   1:  PR[GP1:91,1] = PR[GP1:90,1] + 57.997;
   1:  PR[GP1:91,2] = PR[GP1:90,2] + 23.981;
   1:L PR[91] R[100]mm/sec CNT100;
   1:  PR[GP1:91,1] = PR[GP1:90,1] + 53.597;
   1:  PR[GP1:91,2] = PR[GP1:90,2] + 27.915;
   1:L PR[91] R[100]mm/sec CNT100;
   1:  PR[GP1:91,1] = PR[GP1:90,1] + 52.373;
   1:  PR[GP1:91,2] = PR[GP1:90,2] + 28.903;
   1:L PR[91] R[100]mm/sec CNT100;
   1:  PR[GP1:91,1] = PR[GP1:90,1] + 47.316;
   1:  PR[GP1:91,2] = PR[GP1:90,2] + 32.038;
   1:L PR[91] R[100]mm/sec CNT100;
   1:  PR[GP1:91,1] = PR[GP1:90,1] + 42.338;
   1:  PR[GP1:91,2] = PR[GP1:90,2] + 34.026;
   1:L PR[91] R[100]mm/sec CNT100;
   1:  PR[GP1:91,1] = PR[GP1:90,1] + 39.377;
   1:  PR[GP1:91,2] = PR[GP1:90,2] + 35.072;
   1:L PR[91] R[100]mm/sec CNT100;
   1:  PR[GP1:91,1] = PR[GP1:90,1] + 34.292;
   1:  PR[GP1:91,2] = PR[GP1:90,2] + 36.166;
   1:L PR[91] R[100]mm/sec CNT100;
   1:  PR[GP1:91,1] = PR[GP1:90,1] + 29.702;
   1:  PR[GP1:91,2] = PR[GP1:90,2] + 36.339;
   1:L PR[91] R[100]mm/sec CNT100;
   1:  PR[GP1:91,1] = PR[GP1:90,1] + 24.959;
   1:  PR[GP1:91,2] = PR[GP1:90,2] + 36.356;
   1:L PR[91] R[100]mm/sec CNT100;
   1:  PR[GP1:91,1] = PR[GP1:90,1] + 20.626;
   1:  PR[GP1:91,2] = PR[GP1:90,2] + 35.786;
   1:L PR[91] R[100]mm/sec CNT100;
   1:  PR[GP1:91,1] = PR[GP1:90,1] + 16.906;
   1:  PR[GP1:91,2] = PR[GP1:90,2] + 34.602;
   1:L PR[91] R[100]mm/sec CNT100;
   1:  PR[GP1:91,1] = PR[GP1:90,1] + 11.165;
   1:  PR[GP1:91,2] = PR[GP1:90,2] + 32.612;
   1:L PR[91] R[100]mm/sec CNT100;
   1:  PR[GP1:91,1] = PR[GP1:90,1] + 7.980;
   1:  PR[GP1:91,2] = PR[GP1:90,2] + 30.950;
   1:L PR[91] R[100]mm/sec CNT100;
   1:  PR[GP1:91,1] = PR[GP1:90,1] + 5.211;
   1:  PR[GP1:91,2] = PR[GP1:90,2] + 28.994;
   1:L PR[91] R[100]mm/sec CNT100;
   1:  PR[GP1:91,1] = PR[GP1:90,1] + 4.255;
   1:  PR[GP1:91,2] = PR[GP1:90,2] + 28.246;
   1:L PR[91] R[100]mm/sec CNT100;
   1:  PR[GP1:91,1] = PR[GP1:90,1] + 3.446;
   1:  PR[GP1:91,2] = PR[GP1:90,2] + 27.305;
   1:L PR[91] R[100]mm/sec CNT100;
   1:  PR[GP1:91,1] = PR[GP1:90,1] + 1.713;
   1:  PR[GP1:91,2] = PR[GP1:90,2] + 26.621;
   1:L PR[91] R[100]mm/sec CNT100;
   1:  PR[GP1:91,1] = PR[GP1:90,1] + 1.290;
   1:  PR[GP1:91,2] = PR[GP1:90,2] + 26.404;
   1:L PR[91] R[100]mm/sec CNT100;
   1:  ! -- Layer/Ebene 89 -- !;
   1:  PR[91] = PR[90];
   1:  PR[GP1:91,1] = PR[GP1:90,1] + -2.453;
   1:  PR[GP1:91,2] = PR[GP1:90,2] + 27.220;
   1:  PR[GP1:91,3] = PR[GP1:90,3] + 54.595;
   1:L PR[91] R[100]mm/sec CNT100;
   1:  PR[GP1:91,1] = PR[GP1:90,1] + -3.226;
   1:  PR[GP1:91,2] = PR[GP1:90,2] + 27.613;
   1:L PR[91] R[100]mm/sec CNT100;
   1:  PR[GP1:91,1] = PR[GP1:90,1] + -3.881;
   1:  PR[GP1:91,2] = PR[GP1:90,2] + 28.375;
   1:L PR[91] R[100]mm/sec CNT100;
   1:  PR[GP1:91,1] = PR[GP1:90,1] + -4.669;
   1:  PR[GP1:91,2] = PR[GP1:90,2] + 28.992;
   1:L PR[91] R[100]mm/sec CNT100;
   1:  PR[GP1:91,1] = PR[GP1:90,1] + -7.549;
   1:  PR[GP1:91,2] = PR[GP1:90,2] + 31.027;
   1:L PR[91] R[100]mm/sec CNT100;
   1:  PR[GP1:91,1] = PR[GP1:90,1] + -10.616;
   1:  PR[GP1:91,2] = PR[GP1:90,2] + 32.632;
   1:L PR[91] R[100]mm/sec CNT100;
   1:  PR[GP1:91,1] = PR[GP1:90,1] + -14.394;
   1:  PR[GP1:91,2] = PR[GP1:90,2] + 33.846;
   1:L PR[91] R[100]mm/sec CNT100;
   1:  PR[GP1:91,1] = PR[GP1:90,1] + -20.227;
   1:  PR[GP1:91,2] = PR[GP1:90,2] + 35.862;
   1:L PR[91] R[100]mm/sec CNT100;
   1:  PR[GP1:91,1] = PR[GP1:90,1] + -24.397;
   1:  PR[GP1:91,2] = PR[GP1:90,2] + 36.407;
   1:L PR[91] R[100]mm/sec CNT100;
   1:  PR[GP1:91,1] = PR[GP1:90,1] + -29.289;
   1:  PR[GP1:91,2] = PR[GP1:90,2] + 36.239;
   1:L PR[91] R[100]mm/sec CNT100;
   1:  PR[GP1:91,1] = PR[GP1:90,1] + -33.933;
   1:  PR[GP1:91,2] = PR[GP1:90,2] + 36.216;
   1:L PR[91] R[100]mm/sec CNT100;
   1:  PR[GP1:91,1] = PR[GP1:90,1] + -38.847;
   1:  PR[GP1:91,2] = PR[GP1:90,2] + 35.155;
   1:L PR[91] R[100]mm/sec CNT100;
   1:  PR[GP1:91,1] = PR[GP1:90,1] + -44.230;
   1:  PR[GP1:91,2] = PR[GP1:90,2] + 33.024;
   1:L PR[91] R[100]mm/sec CNT100;
   1:  PR[GP1:91,1] = PR[GP1:90,1] + -46.959;
   1:  PR[GP1:91,2] = PR[GP1:90,2] + 32.055;
   1:L PR[91] R[100]mm/sec CNT100;
   1:  PR[GP1:91,1] = PR[GP1:90,1] + -51.884;
   1:  PR[GP1:91,2] = PR[GP1:90,2] + 28.987;
   1:L PR[91] R[100]mm/sec CNT100;
   1:  PR[GP1:91,1] = PR[GP1:90,1] + -56.664;
   1:  PR[GP1:91,2] = PR[GP1:90,2] + 24.742;
   1:L PR[91] R[100]mm/sec CNT100;
   1:  PR[GP1:91,1] = PR[GP1:90,1] + -57.689;
   1:  PR[GP1:91,2] = PR[GP1:90,2] + 23.913;
   1:L PR[91] R[100]mm/sec CNT100;
   1:  PR[GP1:91,1] = PR[GP1:90,1] + -61.507;
   1:  PR[GP1:91,2] = PR[GP1:90,2] + 18.944;
   1:L PR[91] R[100]mm/sec CNT100;
   1:  PR[GP1:91,1] = PR[GP1:90,1] + -64.708;
   1:  PR[GP1:91,2] = PR[GP1:90,2] + 12.732;
   1:L PR[91] R[100]mm/sec CNT100;
   1:  PR[GP1:91,1] = PR[GP1:90,1] + -64.834;
   1:  PR[GP1:91,2] = PR[GP1:90,2] + 12.522;
   1:L PR[91] R[100]mm/sec CNT100;
   1:  PR[GP1:91,1] = PR[GP1:90,1] + -66.655;
   1:  PR[GP1:91,2] = PR[GP1:90,2] + 6.345;
   1:L PR[91] R[100]mm/sec CNT100;
   1:  PR[GP1:91,1] = PR[GP1:90,1] + -67.234;
   1:  PR[GP1:91,2] = PR[GP1:90,2] + -0.052;
   1:L PR[91] R[100]mm/sec CNT100;
   1:  PR[GP1:91,1] = PR[GP1:90,1] + -67.229;
   1:  PR[GP1:91,2] = PR[GP1:90,2] + -0.083;
   1:L PR[91] R[100]mm/sec CNT100;
   1:  PR[GP1:91,1] = PR[GP1:90,1] + -66.655;
   1:  PR[GP1:91,2] = PR[GP1:90,2] + -6.489;
   1:L PR[91] R[100]mm/sec CNT100;
   1:  PR[GP1:91,1] = PR[GP1:90,1] + -64.828;
   1:  PR[GP1:91,2] = PR[GP1:90,2] + -12.686;
   1:L PR[91] R[100]mm/sec CNT100;
   1:  PR[GP1:91,1] = PR[GP1:90,1] + -61.862;
   1:  PR[GP1:91,2] = PR[GP1:90,2] + -18.501;
   1:L PR[91] R[100]mm/sec CNT100;
   1:  PR[GP1:91,1] = PR[GP1:90,1] + -61.519;
   1:  PR[GP1:91,2] = PR[GP1:90,2] + -19.072;
   1:L PR[91] R[100]mm/sec CNT100;
   1:  PR[GP1:91,1] = PR[GP1:90,1] + -57.679;
   1:  PR[GP1:91,2] = PR[GP1:90,2] + -24.070;
   1:L PR[91] R[100]mm/sec CNT100;
   1:  PR[GP1:91,1] = PR[GP1:90,1] + -53.369;
   1:  PR[GP1:91,2] = PR[GP1:90,2] + -27.936;
   1:L PR[91] R[100]mm/sec CNT100;
   1:  PR[GP1:91,1] = PR[GP1:90,1] + -51.894;
   1:  PR[GP1:91,2] = PR[GP1:90,2] + -29.125;
   1:L PR[91] R[100]mm/sec CNT100;
   1:  PR[GP1:91,1] = PR[GP1:90,1] + -46.946;
   1:  PR[GP1:91,2] = PR[GP1:90,2] + -32.207;
   1:L PR[91] R[100]mm/sec CNT100;
   1:  PR[GP1:91,1] = PR[GP1:90,1] + -42.112;
   1:  PR[GP1:91,2] = PR[GP1:90,2] + -34.148;
   1:L PR[91] R[100]mm/sec CNT100;
   1:  PR[GP1:91,1] = PR[GP1:90,1] + -38.854;
   1:  PR[GP1:91,2] = PR[GP1:90,2] + -35.298;
   1:L PR[91] R[100]mm/sec CNT100;
   1:  PR[GP1:91,1] = PR[GP1:90,1] + -33.917;
   1:  PR[GP1:91,2] = PR[GP1:90,2] + -36.363;
   1:L PR[91] R[100]mm/sec CNT100;
   1:  PR[GP1:91,1] = PR[GP1:90,1] + -29.447;
   1:  PR[GP1:91,2] = PR[GP1:90,2] + -36.535;
   1:L PR[91] R[100]mm/sec CNT100;
   1:  PR[GP1:91,1] = PR[GP1:90,1] + -24.397;
   1:  PR[GP1:91,2] = PR[GP1:90,2] + -36.551;
   1:L PR[91] R[100]mm/sec CNT100;
   1:  PR[GP1:91,1] = PR[GP1:90,1] + -20.210;
   1:  PR[GP1:91,2] = PR[GP1:90,2] + -36.004;
   1:L PR[91] R[100]mm/sec CNT100;
   1:  PR[GP1:91,1] = PR[GP1:90,1] + -16.625;
   1:  PR[GP1:91,2] = PR[GP1:90,2] + -34.863;
   1:L PR[91] R[100]mm/sec CNT100;
   1:  PR[GP1:91,1] = PR[GP1:90,1] + -10.613;
   1:  PR[GP1:91,2] = PR[GP1:90,2] + -32.774;
   1:L PR[91] R[100]mm/sec CNT100;
   1:  PR[GP1:91,1] = PR[GP1:90,1] + -7.546;
   1:  PR[GP1:91,2] = PR[GP1:90,2] + -31.169;
   1:L PR[91] R[100]mm/sec CNT100;
   1:  PR[GP1:91,1] = PR[GP1:90,1] + -3.573;
   1:  PR[GP1:91,2] = PR[GP1:90,2] + -28.282;
   1:L PR[91] R[100]mm/sec CNT100;
   1:  PR[GP1:91,1] = PR[GP1:90,1] + -3.414;
   1:  PR[GP1:91,2] = PR[GP1:90,2] + -28.158;
   1:L PR[91] R[100]mm/sec CNT100;
   1:  PR[GP1:91,1] = PR[GP1:90,1] + -3.168;
   1:  PR[GP1:91,2] = PR[GP1:90,2] + -27.873;
   1:L PR[91] R[100]mm/sec CNT100;
   1:  PR[GP1:91,1] = PR[GP1:90,1] + 0.870;
   1:  PR[GP1:91,2] = PR[GP1:90,2] + -27.006;
   1:L PR[91] R[100]mm/sec CNT100;
   1:  PR[GP1:91,1] = PR[GP1:90,1] + 1.216;
   1:  PR[GP1:91,2] = PR[GP1:90,2] + -26.822;
   1:L PR[91] R[100]mm/sec CNT100;
   1:  PR[GP1:91,1] = PR[GP1:90,1] + 3.432;
   1:  PR[GP1:91,2] = PR[GP1:90,2] + -27.937;
   1:L PR[91] R[100]mm/sec CNT100;
   1:  PR[GP1:91,1] = PR[GP1:90,1] + 3.626;
   1:  PR[GP1:91,2] = PR[GP1:90,2] + -28.162;
   1:L PR[91] R[100]mm/sec CNT100;
   1:  PR[GP1:91,1] = PR[GP1:90,1] + 3.783;
   1:  PR[GP1:91,2] = PR[GP1:90,2] + -28.285;
   1:L PR[91] R[100]mm/sec CNT100;
   1:  PR[GP1:91,1] = PR[GP1:90,1] + 7.766;
   1:  PR[GP1:91,2] = PR[GP1:90,2] + -31.179;
   1:L PR[91] R[100]mm/sec CNT100;
   1:  PR[GP1:91,1] = PR[GP1:90,1] + 10.807;
   1:  PR[GP1:91,2] = PR[GP1:90,2] + -32.766;
   1:L PR[91] R[100]mm/sec CNT100;
   1:  PR[GP1:91,1] = PR[GP1:90,1] + 14.586;
   1:  PR[GP1:91,2] = PR[GP1:90,2] + -33.980;
   1:L PR[91] R[100]mm/sec CNT100;
   1:  PR[GP1:91,1] = PR[GP1:90,1] + 20.426;
   1:  PR[GP1:91,2] = PR[GP1:90,2] + -36.002;
   1:L PR[91] R[100]mm/sec CNT100;
   1:  PR[GP1:91,1] = PR[GP1:90,1] + 24.591;
   1:  PR[GP1:91,2] = PR[GP1:90,2] + -36.549;
   1:L PR[91] R[100]mm/sec CNT100;
   1:  PR[GP1:91,1] = PR[GP1:90,1] + 29.460;
   1:  PR[GP1:91,2] = PR[GP1:90,2] + -36.386;
   1:L PR[91] R[100]mm/sec CNT100;
   1:  PR[GP1:91,1] = PR[GP1:90,1] + 34.110;
   1:  PR[GP1:91,2] = PR[GP1:90,2] + -36.365;
   1:L PR[91] R[100]mm/sec CNT100;
   1:  PR[GP1:91,1] = PR[GP1:90,1] + 39.017;
   1:  PR[GP1:91,2] = PR[GP1:90,2] + -35.309;
   1:L PR[91] R[100]mm/sec CNT100;
   1:  PR[GP1:91,1] = PR[GP1:90,1] + 44.407;
   1:  PR[GP1:91,2] = PR[GP1:90,2] + -33.186;
   1:L PR[91] R[100]mm/sec CNT100;
   1:  PR[GP1:91,1] = PR[GP1:90,1] + 47.142;
   1:  PR[GP1:91,2] = PR[GP1:90,2] + -32.216;
   1:L PR[91] R[100]mm/sec CNT100;
   1:  PR[GP1:91,1] = PR[GP1:90,1] + 52.036;
   1:  PR[GP1:91,2] = PR[GP1:90,2] + -29.183;
   1:L PR[91] R[100]mm/sec CNT100;
   1:  PR[GP1:91,1] = PR[GP1:90,1] + 56.791;
   1:  PR[GP1:91,2] = PR[GP1:90,2] + -24.972;
   1:L PR[91] R[100]mm/sec CNT100;
   1:  PR[GP1:91,1] = PR[GP1:90,1] + 57.825;
   1:  PR[GP1:91,2] = PR[GP1:90,2] + -24.135;
   1:L PR[91] R[100]mm/sec CNT100;
   1:  PR[GP1:91,1] = PR[GP1:90,1] + 61.682;
   1:  PR[GP1:91,2] = PR[GP1:90,2] + -19.128;
   1:L PR[91] R[100]mm/sec CNT100;
   1:  PR[GP1:91,1] = PR[GP1:90,1] + 64.892;
   1:  PR[GP1:91,2] = PR[GP1:90,2] + -12.967;
   1:L PR[91] R[100]mm/sec CNT100;
   1:  PR[GP1:91,1] = PR[GP1:90,1] + 65.020;
   1:  PR[GP1:91,2] = PR[GP1:90,2] + -12.754;
   1:L PR[91] R[100]mm/sec CNT100;
   1:  PR[GP1:91,1] = PR[GP1:90,1] + 66.839;
   1:  PR[GP1:91,2] = PR[GP1:90,2] + -6.669;
   1:L PR[91] R[100]mm/sec CNT100;
   1:  PR[GP1:91,1] = PR[GP1:90,1] + 67.449;
   1:  PR[GP1:91,2] = PR[GP1:90,2] + -0.072;
   1:L PR[91] R[100]mm/sec CNT100;
   1:  PR[GP1:91,1] = PR[GP1:90,1] + 66.839;
   1:  PR[GP1:91,2] = PR[GP1:90,2] + 6.525;
   1:L PR[91] R[100]mm/sec CNT100;
   1:  PR[GP1:91,1] = PR[GP1:90,1] + 65.015;
   1:  PR[GP1:91,2] = PR[GP1:90,2] + 12.629;
   1:L PR[91] R[100]mm/sec CNT100;
   1:  PR[GP1:91,1] = PR[GP1:90,1] + 62.040;
   1:  PR[GP1:91,2] = PR[GP1:90,2] + 18.394;
   1:L PR[91] R[100]mm/sec CNT100;
   1:  PR[GP1:91,1] = PR[GP1:90,1] + 61.694;
   1:  PR[GP1:91,2] = PR[GP1:90,2] + 18.969;
   1:L PR[91] R[100]mm/sec CNT100;
   1:  PR[GP1:91,1] = PR[GP1:90,1] + 57.816;
   1:  PR[GP1:91,2] = PR[GP1:90,2] + 24.003;
   1:L PR[91] R[100]mm/sec CNT100;
   1:  PR[GP1:91,1] = PR[GP1:90,1] + 53.529;
   1:  PR[GP1:91,2] = PR[GP1:90,2] + 27.836;
   1:L PR[91] R[100]mm/sec CNT100;
   1:  PR[GP1:91,1] = PR[GP1:90,1] + 52.050;
   1:  PR[GP1:91,2] = PR[GP1:90,2] + 29.030;
   1:L PR[91] R[100]mm/sec CNT100;
   1:  PR[GP1:91,1] = PR[GP1:90,1] + 47.134;
   1:  PR[GP1:91,2] = PR[GP1:90,2] + 32.078;
   1:L PR[91] R[100]mm/sec CNT100;
   1:  PR[GP1:91,1] = PR[GP1:90,1] + 42.293;
   1:  PR[GP1:91,2] = PR[GP1:90,2] + 34.011;
   1:L PR[91] R[100]mm/sec CNT100;
   1:  PR[GP1:91,1] = PR[GP1:90,1] + 39.032;
   1:  PR[GP1:91,2] = PR[GP1:90,2] + 35.162;
   1:L PR[91] R[100]mm/sec CNT100;
   1:  PR[GP1:91,1] = PR[GP1:90,1] + 34.105;
   1:  PR[GP1:91,2] = PR[GP1:90,2] + 36.222;
   1:L PR[91] R[100]mm/sec CNT100;
   1:  PR[GP1:91,1] = PR[GP1:90,1] + 29.656;
   1:  PR[GP1:91,2] = PR[GP1:90,2] + 36.390;
   1:L PR[91] R[100]mm/sec CNT100;
   1:  PR[GP1:91,1] = PR[GP1:90,1] + 24.608;
   1:  PR[GP1:91,2] = PR[GP1:90,2] + 36.408;
   1:L PR[91] R[100]mm/sec CNT100;
   1:  PR[GP1:91,1] = PR[GP1:90,1] + 20.428;
   1:  PR[GP1:91,2] = PR[GP1:90,2] + 35.858;
   1:L PR[91] R[100]mm/sec CNT100;
   1:  PR[GP1:91,1] = PR[GP1:90,1] + 16.838;
   1:  PR[GP1:91,2] = PR[GP1:90,2] + 34.716;
   1:L PR[91] R[100]mm/sec CNT100;
   1:  PR[GP1:91,1] = PR[GP1:90,1] + 10.823;
   1:  PR[GP1:91,2] = PR[GP1:90,2] + 32.631;
   1:L PR[91] R[100]mm/sec CNT100;
   1:  PR[GP1:91,1] = PR[GP1:90,1] + 7.768;
   1:  PR[GP1:91,2] = PR[GP1:90,2] + 31.037;
   1:L PR[91] R[100]mm/sec CNT100;
   1:  PR[GP1:91,1] = PR[GP1:90,1] + 4.881;
   1:  PR[GP1:91,2] = PR[GP1:90,2] + 28.997;
   1:L PR[91] R[100]mm/sec CNT100;
   1:  PR[GP1:91,1] = PR[GP1:90,1] + 4.097;
   1:  PR[GP1:91,2] = PR[GP1:90,2] + 28.384;
   1:L PR[91] R[100]mm/sec CNT100;
   1:  PR[GP1:91,1] = PR[GP1:90,1] + 3.417;
   1:  PR[GP1:91,2] = PR[GP1:90,2] + 27.592;
   1:L PR[91] R[100]mm/sec CNT100;
   1:  PR[GP1:91,1] = PR[GP1:90,1] + 1.625;
   1:  PR[GP1:91,2] = PR[GP1:90,2] + 26.884;
   1:L PR[91] R[100]mm/sec CNT100;
   1:  PR[GP1:91,1] = PR[GP1:90,1] + 1.331;
   1:  PR[GP1:91,2] = PR[GP1:90,2] + 26.734;
   1:L PR[91] R[100]mm/sec CNT100;
   1:  ! -- Layer/Ebene 90 -- !;
   1:  PR[91] = PR[90];
   1:  PR[GP1:91,1] = PR[GP1:90,1] + -2.542;
   1:  PR[GP1:91,2] = PR[GP1:90,2] + 27.567;
   1:  PR[GP1:91,3] = PR[GP1:90,3] + 55.205;
   1:L PR[91] R[100]mm/sec CNT100;
   1:  PR[GP1:91,1] = PR[GP1:90,1] + -3.196;
   1:  PR[GP1:91,2] = PR[GP1:90,2] + 27.900;
   1:L PR[91] R[100]mm/sec CNT100;
   1:  PR[GP1:91,1] = PR[GP1:90,1] + -3.725;
   1:  PR[GP1:91,2] = PR[GP1:90,2] + 28.515;
   1:L PR[91] R[100]mm/sec CNT100;
   1:  PR[GP1:91,1] = PR[GP1:90,1] + -4.339;
   1:  PR[GP1:91,2] = PR[GP1:90,2] + 28.995;
   1:L PR[91] R[100]mm/sec CNT100;
   1:  PR[GP1:91,1] = PR[GP1:90,1] + -7.338;
   1:  PR[GP1:91,2] = PR[GP1:90,2] + 31.114;
   1:L PR[91] R[100]mm/sec CNT100;
   1:  PR[GP1:91,1] = PR[GP1:90,1] + -10.275;
   1:  PR[GP1:91,2] = PR[GP1:90,2] + 32.651;
   1:L PR[91] R[100]mm/sec CNT100;
   1:  PR[GP1:91,1] = PR[GP1:90,1] + -13.893;
   1:  PR[GP1:91,2] = PR[GP1:90,2] + 33.814;
   1:L PR[91] R[100]mm/sec CNT100;
   1:  PR[GP1:91,1] = PR[GP1:90,1] + -20.028;
   1:  PR[GP1:91,2] = PR[GP1:90,2] + 35.934;
   1:L PR[91] R[100]mm/sec CNT100;
   1:  PR[GP1:91,1] = PR[GP1:90,1] + -24.045;
   1:  PR[GP1:91,2] = PR[GP1:90,2] + 36.459;
   1:L PR[91] R[100]mm/sec CNT100;
   1:  PR[GP1:91,1] = PR[GP1:90,1] + -28.760;
   1:  PR[GP1:91,2] = PR[GP1:90,2] + 36.297;
   1:L PR[91] R[100]mm/sec CNT100;
   1:  PR[GP1:91,1] = PR[GP1:90,1] + -33.745;
   1:  PR[GP1:91,2] = PR[GP1:90,2] + 36.272;
   1:L PR[91] R[100]mm/sec CNT100;
   1:  PR[GP1:91,1] = PR[GP1:90,1] + -38.502;
   1:  PR[GP1:91,2] = PR[GP1:90,2] + 35.246;
   1:L PR[91] R[100]mm/sec CNT100;
   1:  PR[GP1:91,1] = PR[GP1:90,1] + -43.714;
   1:  PR[GP1:91,2] = PR[GP1:90,2] + 33.182;
   1:L PR[91] R[100]mm/sec CNT100;
   1:  PR[GP1:91,1] = PR[GP1:90,1] + -46.775;
   1:  PR[GP1:91,2] = PR[GP1:90,2] + 32.095;
   1:L PR[91] R[100]mm/sec CNT100;
   1:  PR[GP1:91,1] = PR[GP1:90,1] + -51.559;
   1:  PR[GP1:91,2] = PR[GP1:90,2] + 29.116;
   1:L PR[91] R[100]mm/sec CNT100;
   1:  PR[GP1:91,1] = PR[GP1:90,1] + -56.204;
   1:  PR[GP1:91,2] = PR[GP1:90,2] + 24.991;
   1:L PR[91] R[100]mm/sec CNT100;
   1:  PR[GP1:91,1] = PR[GP1:90,1] + -57.506;
   1:  PR[GP1:91,2] = PR[GP1:90,2] + 23.937;
   1:L PR[91] R[100]mm/sec CNT100;
   1:  PR[GP1:91,1] = PR[GP1:90,1] + -61.222;
   1:  PR[GP1:91,2] = PR[GP1:90,2] + 19.100;
   1:L PR[91] R[100]mm/sec CNT100;
   1:  PR[GP1:91,1] = PR[GP1:90,1] + -64.340;
   1:  PR[GP1:91,2] = PR[GP1:90,2] + 13.051;
   1:L PR[91] R[100]mm/sec CNT100;
   1:  PR[GP1:91,1] = PR[GP1:90,1] + -64.647;
   1:  PR[GP1:91,2] = PR[GP1:90,2] + 12.538;
   1:L PR[91] R[100]mm/sec CNT100;
   1:  PR[GP1:91,1] = PR[GP1:90,1] + -66.422;
   1:  PR[GP1:91,2] = PR[GP1:90,2] + 6.516;
   1:L PR[91] R[100]mm/sec CNT100;
   1:  PR[GP1:91,1] = PR[GP1:90,1] + -67.006;
   1:  PR[GP1:91,2] = PR[GP1:90,2] + 0.129;
   1:L PR[91] R[100]mm/sec CNT100;
   1:  PR[GP1:91,1] = PR[GP1:90,1] + -67.048;
   1:  PR[GP1:91,2] = PR[GP1:90,2] + -0.100;
   1:L PR[91] R[100]mm/sec CNT100;
   1:  PR[GP1:91,1] = PR[GP1:90,1] + -66.485;
   1:  PR[GP1:91,2] = PR[GP1:90,2] + -6.334;
   1:L PR[91] R[100]mm/sec CNT100;
   1:  PR[GP1:91,1] = PR[GP1:90,1] + -66.430;
   1:  PR[GP1:91,2] = PR[GP1:90,2] + -6.634;
   1:L PR[91] R[100]mm/sec CNT100;
   1:  PR[GP1:91,1] = PR[GP1:90,1] + -64.641;
   1:  PR[GP1:91,2] = PR[GP1:90,2] + -12.701;
   1:L PR[91] R[100]mm/sec CNT100;
   1:  PR[GP1:91,1] = PR[GP1:90,1] + -61.749;
   1:  PR[GP1:91,2] = PR[GP1:90,2] + -18.372;
   1:L PR[91] R[100]mm/sec CNT100;
   1:  PR[GP1:91,1] = PR[GP1:90,1] + -61.234;
   1:  PR[GP1:91,2] = PR[GP1:90,2] + -19.229;
   1:L PR[91] R[100]mm/sec CNT100;
   1:  PR[GP1:91,1] = PR[GP1:90,1] + -57.496;
   1:  PR[GP1:91,2] = PR[GP1:90,2] + -24.094;
   1:L PR[91] R[100]mm/sec CNT100;
   1:  PR[GP1:91,1] = PR[GP1:90,1] + -53.299;
   1:  PR[GP1:91,2] = PR[GP1:90,2] + -27.859;
   1:L PR[91] R[100]mm/sec CNT100;
   1:  PR[GP1:91,1] = PR[GP1:90,1] + -51.569;
   1:  PR[GP1:91,2] = PR[GP1:90,2] + -29.253;
   1:L PR[91] R[100]mm/sec CNT100;
   1:  PR[GP1:91,1] = PR[GP1:90,1] + -46.763;
   1:  PR[GP1:91,2] = PR[GP1:90,2] + -32.247;
   1:L PR[91] R[100]mm/sec CNT100;
   1:  PR[GP1:91,1] = PR[GP1:90,1] + -42.067;
   1:  PR[GP1:91,2] = PR[GP1:90,2] + -34.133;
   1:L PR[91] R[100]mm/sec CNT100;
   1:  PR[GP1:91,1] = PR[GP1:90,1] + -38.508;
   1:  PR[GP1:91,2] = PR[GP1:90,2] + -35.389;
   1:L PR[91] R[100]mm/sec CNT100;
   1:  PR[GP1:91,1] = PR[GP1:90,1] + -33.729;
   1:  PR[GP1:91,2] = PR[GP1:90,2] + -36.419;
   1:L PR[91] R[100]mm/sec CNT100;
   1:  PR[GP1:91,1] = PR[GP1:90,1] + -29.401;
   1:  PR[GP1:91,2] = PR[GP1:90,2] + -36.586;
   1:L PR[91] R[100]mm/sec CNT100;
   1:  PR[GP1:91,1] = PR[GP1:90,1] + -24.045;
   1:  PR[GP1:91,2] = PR[GP1:90,2] + -36.603;
   1:L PR[91] R[100]mm/sec CNT100;
   1:  PR[GP1:91,1] = PR[GP1:90,1] + -20.011;
   1:  PR[GP1:91,2] = PR[GP1:90,2] + -36.076;
   1:L PR[91] R[100]mm/sec CNT100;
   1:  PR[GP1:91,1] = PR[GP1:90,1] + -16.557;
   1:  PR[GP1:91,2] = PR[GP1:90,2] + -34.977;
   1:L PR[91] R[100]mm/sec CNT100;
   1:  PR[GP1:91,1] = PR[GP1:90,1] + -10.270;
   1:  PR[GP1:91,2] = PR[GP1:90,2] + -32.792;
   1:L PR[91] R[100]mm/sec CNT100;
   1:  PR[GP1:91,1] = PR[GP1:90,1] + -7.335;
   1:  PR[GP1:91,2] = PR[GP1:90,2] + -31.256;
   1:L PR[91] R[100]mm/sec CNT100;
   1:  PR[GP1:91,1] = PR[GP1:90,1] + -3.067;
   1:  PR[GP1:91,2] = PR[GP1:90,2] + -28.151;
   1:L PR[91] R[100]mm/sec CNT100;
   1:  PR[GP1:91,1] = PR[GP1:90,1] + 1.345;
   1:  PR[GP1:91,2] = PR[GP1:90,2] + -27.196;
   1:L PR[91] R[100]mm/sec CNT100;
   1:  PR[GP1:91,1] = PR[GP1:90,1] + 3.338;
   1:  PR[GP1:91,2] = PR[GP1:90,2] + -28.198;
   1:L PR[91] R[100]mm/sec CNT100;
   1:  PR[GP1:91,1] = PR[GP1:90,1] + 7.554;
   1:  PR[GP1:91,2] = PR[GP1:90,2] + -31.265;
   1:L PR[91] R[100]mm/sec CNT100;
   1:  PR[GP1:91,1] = PR[GP1:90,1] + 10.465;
   1:  PR[GP1:91,2] = PR[GP1:90,2] + -32.784;
   1:L PR[91] R[100]mm/sec CNT100;
   1:  PR[GP1:91,1] = PR[GP1:90,1] + 14.085;
   1:  PR[GP1:91,2] = PR[GP1:90,2] + -33.947;
   1:L PR[91] R[100]mm/sec CNT100;
   1:  PR[GP1:91,1] = PR[GP1:90,1] + 20.227;
   1:  PR[GP1:91,2] = PR[GP1:90,2] + -36.074;
   1:L PR[91] R[100]mm/sec CNT100;
   1:  PR[GP1:91,1] = PR[GP1:90,1] + 24.239;
   1:  PR[GP1:91,2] = PR[GP1:90,2] + -36.602;
   1:L PR[91] R[100]mm/sec CNT100;
   1:  PR[GP1:91,1] = PR[GP1:90,1] + 28.932;
   1:  PR[GP1:91,2] = PR[GP1:90,2] + -36.444;
   1:L PR[91] R[100]mm/sec CNT100;
   1:  PR[GP1:91,1] = PR[GP1:90,1] + 33.922;
   1:  PR[GP1:91,2] = PR[GP1:90,2] + -36.422;
   1:L PR[91] R[100]mm/sec CNT100;
   1:  PR[GP1:91,1] = PR[GP1:90,1] + 38.672;
   1:  PR[GP1:91,2] = PR[GP1:90,2] + -35.400;
   1:L PR[91] R[100]mm/sec CNT100;
   1:  PR[GP1:91,1] = PR[GP1:90,1] + 43.892;
   1:  PR[GP1:91,2] = PR[GP1:90,2] + -33.343;
   1:L PR[91] R[100]mm/sec CNT100;
   1:  PR[GP1:91,1] = PR[GP1:90,1] + 46.959;
   1:  PR[GP1:91,2] = PR[GP1:90,2] + -32.256;
   1:L PR[91] R[100]mm/sec CNT100;
   1:  PR[GP1:91,1] = PR[GP1:90,1] + 51.713;
   1:  PR[GP1:91,2] = PR[GP1:90,2] + -29.309;
   1:L PR[91] R[100]mm/sec CNT100;
   1:  PR[GP1:91,1] = PR[GP1:90,1] + 56.332;
   1:  PR[GP1:91,2] = PR[GP1:90,2] + -25.219;
   1:L PR[91] R[100]mm/sec CNT100;
   1:  PR[GP1:91,1] = PR[GP1:90,1] + 57.643;
   1:  PR[GP1:91,2] = PR[GP1:90,2] + -24.158;
   1:L PR[91] R[100]mm/sec CNT100;
   1:  PR[GP1:91,1] = PR[GP1:90,1] + 61.398;
   1:  PR[GP1:91,2] = PR[GP1:90,2] + -19.283;
   1:L PR[91] R[100]mm/sec CNT100;
   1:  PR[GP1:91,1] = PR[GP1:90,1] + 64.525;
   1:  PR[GP1:91,2] = PR[GP1:90,2] + -13.283;
   1:L PR[91] R[100]mm/sec CNT100;
   1:  PR[GP1:91,1] = PR[GP1:90,1] + 64.834;
   1:  PR[GP1:91,2] = PR[GP1:90,2] + -12.768;
   1:L PR[91] R[100]mm/sec CNT100;
   1:  PR[GP1:91,1] = PR[GP1:90,1] + 66.606;
   1:  PR[GP1:91,2] = PR[GP1:90,2] + -6.836;
   1:L PR[91] R[100]mm/sec CNT100;
   1:  PR[GP1:91,1] = PR[GP1:90,1] + 67.220;
   1:  PR[GP1:91,2] = PR[GP1:90,2] + -0.273;
   1:L PR[91] R[100]mm/sec CNT100;
   1:  PR[GP1:91,1] = PR[GP1:90,1] + 67.262;
   1:  PR[GP1:91,2] = PR[GP1:90,2] + -0.045;
   1:L PR[91] R[100]mm/sec CNT100;
   1:  PR[GP1:91,1] = PR[GP1:90,1] + 66.670;
   1:  PR[GP1:91,2] = PR[GP1:90,2] + 6.363;
   1:L PR[91] R[100]mm/sec CNT100;
   1:  PR[GP1:91,1] = PR[GP1:90,1] + 66.614;
   1:  PR[GP1:91,2] = PR[GP1:90,2] + 6.666;
   1:L PR[91] R[100]mm/sec CNT100;
   1:  PR[GP1:91,1] = PR[GP1:90,1] + 64.828;
   1:  PR[GP1:91,2] = PR[GP1:90,2] + 12.643;
   1:L PR[91] R[100]mm/sec CNT100;
   1:  PR[GP1:91,1] = PR[GP1:90,1] + 61.928;
   1:  PR[GP1:91,2] = PR[GP1:90,2] + 18.264;
   1:L PR[91] R[100]mm/sec CNT100;
   1:  PR[GP1:91,1] = PR[GP1:90,1] + 61.410;
   1:  PR[GP1:91,2] = PR[GP1:90,2] + 19.124;
   1:L PR[91] R[100]mm/sec CNT100;
   1:  PR[GP1:91,1] = PR[GP1:90,1] + 57.635;
   1:  PR[GP1:91,2] = PR[GP1:90,2] + 24.025;
   1:L PR[91] R[100]mm/sec CNT100;
   1:  PR[GP1:91,1] = PR[GP1:90,1] + 53.460;
   1:  PR[GP1:91,2] = PR[GP1:90,2] + 27.757;
   1:L PR[91] R[100]mm/sec CNT100;
   1:  PR[GP1:91,1] = PR[GP1:90,1] + 51.726;
   1:  PR[GP1:91,2] = PR[GP1:90,2] + 29.157;
   1:L PR[91] R[100]mm/sec CNT100;
   1:  PR[GP1:91,1] = PR[GP1:90,1] + 46.951;
   1:  PR[GP1:91,2] = PR[GP1:90,2] + 32.117;
   1:L PR[91] R[100]mm/sec CNT100;
   1:  PR[GP1:91,1] = PR[GP1:90,1] + 42.249;
   1:  PR[GP1:91,2] = PR[GP1:90,2] + 33.995;
   1:L PR[91] R[100]mm/sec CNT100;
   1:  PR[GP1:91,1] = PR[GP1:90,1] + 38.688;
   1:  PR[GP1:91,2] = PR[GP1:90,2] + 35.252;
   1:L PR[91] R[100]mm/sec CNT100;
   1:  PR[GP1:91,1] = PR[GP1:90,1] + 33.918;
   1:  PR[GP1:91,2] = PR[GP1:90,2] + 36.279;
   1:L PR[91] R[100]mm/sec CNT100;
   1:  PR[GP1:91,1] = PR[GP1:90,1] + 29.611;
   1:  PR[GP1:91,2] = PR[GP1:90,2] + 36.441;
   1:L PR[91] R[100]mm/sec CNT100;
   1:  PR[GP1:91,1] = PR[GP1:90,1] + 24.257;
   1:  PR[GP1:91,2] = PR[GP1:90,2] + 36.460;
   1:L PR[91] R[100]mm/sec CNT100;
   1:  PR[GP1:91,1] = PR[GP1:90,1] + 20.229;
   1:  PR[GP1:91,2] = PR[GP1:90,2] + 35.931;
   1:L PR[91] R[100]mm/sec CNT100;
   1:  PR[GP1:91,1] = PR[GP1:90,1] + 16.770;
   1:  PR[GP1:91,2] = PR[GP1:90,2] + 34.830;
   1:L PR[91] R[100]mm/sec CNT100;
   1:  PR[GP1:91,1] = PR[GP1:90,1] + 10.482;
   1:  PR[GP1:91,2] = PR[GP1:90,2] + 32.650;
   1:L PR[91] R[100]mm/sec CNT100;
   1:  PR[GP1:91,1] = PR[GP1:90,1] + 7.557;
   1:  PR[GP1:91,2] = PR[GP1:90,2] + 31.124;
   1:L PR[91] R[100]mm/sec CNT100;
   1:  PR[GP1:91,1] = PR[GP1:90,1] + 4.550;
   1:  PR[GP1:91,2] = PR[GP1:90,2] + 28.999;
   1:L PR[91] R[100]mm/sec CNT100;
   1:  PR[GP1:91,1] = PR[GP1:90,1] + 3.939;
   1:  PR[GP1:91,2] = PR[GP1:90,2] + 28.522;
   1:L PR[91] R[100]mm/sec CNT100;
   1:  PR[GP1:91,1] = PR[GP1:90,1] + 3.387;
   1:  PR[GP1:91,2] = PR[GP1:90,2] + 27.879;
   1:L PR[91] R[100]mm/sec CNT100;
   1:  PR[GP1:91,1] = PR[GP1:90,1] + 1.342;
   1:  PR[GP1:91,2] = PR[GP1:90,2] + 27.068;
   1:L PR[91] R[100]mm/sec CNT100;
   1:  ! -- Layer/Ebene 91 -- !;
   1:  PR[91] = PR[90];
   1:  PR[GP1:91,1] = PR[GP1:90,1] + 1.056;
   1:  PR[GP1:91,2] = PR[GP1:90,2] + 27.360;
   1:  PR[GP1:91,3] = PR[GP1:90,3] + 55.815;
   1:L PR[91] R[100]mm/sec CNT100;
   1:  PR[GP1:91,1] = PR[GP1:90,1] + 0.284;
   1:  PR[GP1:91,2] = PR[GP1:90,2] + 27.539;
   1:L PR[91] R[100]mm/sec CNT100;
   1:  PR[GP1:91,1] = PR[GP1:90,1] + -2.631;
   1:  PR[GP1:91,2] = PR[GP1:90,2] + 27.914;
   1:L PR[91] R[100]mm/sec CNT100;
   1:  PR[GP1:91,1] = PR[GP1:90,1] + -3.167;
   1:  PR[GP1:91,2] = PR[GP1:90,2] + 28.187;
   1:L PR[91] R[100]mm/sec CNT100;
   1:  PR[GP1:91,1] = PR[GP1:90,1] + -3.569;
   1:  PR[GP1:91,2] = PR[GP1:90,2] + 28.654;
   1:L PR[91] R[100]mm/sec CNT100;
   1:  PR[GP1:91,1] = PR[GP1:90,1] + -4.009;
   1:  PR[GP1:91,2] = PR[GP1:90,2] + 28.999;
   1:L PR[91] R[100]mm/sec CNT100;
   1:  PR[GP1:91,1] = PR[GP1:90,1] + -7.127;
   1:  PR[GP1:91,2] = PR[GP1:90,2] + 31.202;
   1:L PR[91] R[100]mm/sec CNT100;
   1:  PR[GP1:91,1] = PR[GP1:90,1] + -9.933;
   1:  PR[GP1:91,2] = PR[GP1:90,2] + 32.670;
   1:L PR[91] R[100]mm/sec CNT100;
   1:  PR[GP1:91,1] = PR[GP1:90,1] + -13.393;
   1:  PR[GP1:91,2] = PR[GP1:90,2] + 33.781;
   1:L PR[91] R[100]mm/sec CNT100;
   1:  PR[GP1:91,1] = PR[GP1:90,1] + -19.830;
   1:  PR[GP1:91,2] = PR[GP1:90,2] + 36.007;
   1:L PR[91] R[100]mm/sec CNT100;
   1:  PR[GP1:91,1] = PR[GP1:90,1] + -23.694;
   1:  PR[GP1:91,2] = PR[GP1:90,2] + 36.512;
   1:L PR[91] R[100]mm/sec CNT100;
   1:  PR[GP1:91,1] = PR[GP1:90,1] + -28.232;
   1:  PR[GP1:91,2] = PR[GP1:90,2] + 36.356;
   1:L PR[91] R[100]mm/sec CNT100;
   1:  PR[GP1:91,1] = PR[GP1:90,1] + -33.557;
   1:  PR[GP1:91,2] = PR[GP1:90,2] + 36.329;
   1:L PR[91] R[100]mm/sec CNT100;
   1:  PR[GP1:91,1] = PR[GP1:90,1] + -38.156;
   1:  PR[GP1:91,2] = PR[GP1:90,2] + 35.337;
   1:L PR[91] R[100]mm/sec CNT100;
   1:  PR[GP1:91,1] = PR[GP1:90,1] + -43.198;
   1:  PR[GP1:91,2] = PR[GP1:90,2] + 33.340;
   1:L PR[91] R[100]mm/sec CNT100;
   1:  PR[GP1:91,1] = PR[GP1:90,1] + -46.592;
   1:  PR[GP1:91,2] = PR[GP1:90,2] + 32.135;
   1:L PR[91] R[100]mm/sec CNT100;
   1:  PR[GP1:91,1] = PR[GP1:90,1] + -51.234;
   1:  PR[GP1:91,2] = PR[GP1:90,2] + 29.244;
   1:L PR[91] R[100]mm/sec CNT100;
   1:  PR[GP1:91,1] = PR[GP1:90,1] + -55.744;
   1:  PR[GP1:91,2] = PR[GP1:90,2] + 25.239;
   1:L PR[91] R[100]mm/sec CNT100;
   1:  PR[GP1:91,1] = PR[GP1:90,1] + -57.323;
   1:  PR[GP1:91,2] = PR[GP1:90,2] + 23.961;
   1:L PR[91] R[100]mm/sec CNT100;
   1:  PR[GP1:91,1] = PR[GP1:90,1] + -60.938;
   1:  PR[GP1:91,2] = PR[GP1:90,2] + 19.256;
   1:L PR[91] R[100]mm/sec CNT100;
   1:  PR[GP1:91,1] = PR[GP1:90,1] + -63.972;
   1:  PR[GP1:91,2] = PR[GP1:90,2] + 13.369;
   1:L PR[91] R[100]mm/sec CNT100;
   1:  PR[GP1:91,1] = PR[GP1:90,1] + -64.460;
   1:  PR[GP1:91,2] = PR[GP1:90,2] + 12.553;
   1:L PR[91] R[100]mm/sec CNT100;
   1:  PR[GP1:91,1] = PR[GP1:90,1] + -66.189;
   1:  PR[GP1:91,2] = PR[GP1:90,2] + 6.688;
   1:L PR[91] R[100]mm/sec CNT100;
   1:  PR[GP1:91,1] = PR[GP1:90,1] + -66.758;
   1:  PR[GP1:91,2] = PR[GP1:90,2] + 0.464;
   1:L PR[91] R[100]mm/sec CNT100;
   1:  PR[GP1:91,1] = PR[GP1:90,1] + -66.862;
   1:  PR[GP1:91,2] = PR[GP1:90,2] + -0.100;
   1:L PR[91] R[100]mm/sec CNT100;
   1:  PR[GP1:91,1] = PR[GP1:90,1] + -66.313;
   1:  PR[GP1:91,2] = PR[GP1:90,2] + -6.178;
   1:L PR[91] R[100]mm/sec CNT100;
   1:  PR[GP1:91,1] = PR[GP1:90,1] + -66.197;
   1:  PR[GP1:91,2] = PR[GP1:90,2] + -6.805;
   1:L PR[91] R[100]mm/sec CNT100;
   1:  PR[GP1:91,1] = PR[GP1:90,1] + -64.454;
   1:  PR[GP1:91,2] = PR[GP1:90,2] + -12.717;
   1:L PR[91] R[100]mm/sec CNT100;
   1:  PR[GP1:91,1] = PR[GP1:90,1] + -61.636;
   1:  PR[GP1:91,2] = PR[GP1:90,2] + -18.242;
   1:L PR[91] R[100]mm/sec CNT100;
   1:  PR[GP1:91,1] = PR[GP1:90,1] + -60.949;
   1:  PR[GP1:91,2] = PR[GP1:90,2] + -19.385;
   1:L PR[91] R[100]mm/sec CNT100;
   1:  PR[GP1:91,1] = PR[GP1:90,1] + -57.312;
   1:  PR[GP1:91,2] = PR[GP1:90,2] + -24.119;
   1:L PR[91] R[100]mm/sec CNT100;
   1:  PR[GP1:91,1] = PR[GP1:90,1] + -53.229;
   1:  PR[GP1:91,2] = PR[GP1:90,2] + -27.782;
   1:L PR[91] R[100]mm/sec CNT100;
   1:  PR[GP1:91,1] = PR[GP1:90,1] + -51.244;
   1:  PR[GP1:91,2] = PR[GP1:90,2] + -29.381;
   1:L PR[91] R[100]mm/sec CNT100;
   1:  PR[GP1:91,1] = PR[GP1:90,1] + -46.579;
   1:  PR[GP1:91,2] = PR[GP1:90,2] + -32.287;
   1:L PR[91] R[100]mm/sec CNT100;
   1:  PR[GP1:91,1] = PR[GP1:90,1] + -42.021;
   1:  PR[GP1:91,2] = PR[GP1:90,2] + -34.118;
   1:L PR[91] R[100]mm/sec CNT100;
   1:  PR[GP1:91,1] = PR[GP1:90,1] + -38.162;
   1:  PR[GP1:91,2] = PR[GP1:90,2] + -35.479;
   1:L PR[91] R[100]mm/sec CNT100;
   1:  PR[GP1:91,1] = PR[GP1:90,1] + -33.541;
   1:  PR[GP1:91,2] = PR[GP1:90,2] + -36.476;
   1:L PR[91] R[100]mm/sec CNT100;
   1:  PR[GP1:91,1] = PR[GP1:90,1] + -29.355;
   1:  PR[GP1:91,2] = PR[GP1:90,2] + -36.637;
   1:L PR[91] R[100]mm/sec CNT100;
   1:  PR[GP1:91,1] = PR[GP1:90,1] + -23.693;
   1:  PR[GP1:91,2] = PR[GP1:90,2] + -36.655;
   1:L PR[91] R[100]mm/sec CNT100;
   1:  PR[GP1:91,1] = PR[GP1:90,1] + -19.812;
   1:  PR[GP1:91,2] = PR[GP1:90,2] + -36.148;
   1:L PR[91] R[100]mm/sec CNT100;
   1:  PR[GP1:91,1] = PR[GP1:90,1] + -16.488;
   1:  PR[GP1:91,2] = PR[GP1:90,2] + -35.090;
   1:L PR[91] R[100]mm/sec CNT100;
   1:  PR[GP1:91,1] = PR[GP1:90,1] + -9.928;
   1:  PR[GP1:91,2] = PR[GP1:90,2] + -32.811;
   1:L PR[91] R[100]mm/sec CNT100;
   1:  PR[GP1:91,1] = PR[GP1:90,1] + -7.124;
   1:  PR[GP1:91,2] = PR[GP1:90,2] + -31.343;
   1:L PR[91] R[100]mm/sec CNT100;
   1:  PR[GP1:91,1] = PR[GP1:90,1] + -2.994;
   1:  PR[GP1:91,2] = PR[GP1:90,2] + -28.343;
   1:L PR[91] R[100]mm/sec CNT100;
   1:  PR[GP1:91,1] = PR[GP1:90,1] + -2.734;
   1:  PR[GP1:91,2] = PR[GP1:90,2] + -28.332;
   1:L PR[91] R[100]mm/sec CNT100;
   1:  PR[GP1:91,1] = PR[GP1:90,1] + 1.378;
   1:  PR[GP1:91,2] = PR[GP1:90,2] + -27.455;
   1:L PR[91] R[100]mm/sec CNT100;
   1:  PR[GP1:91,1] = PR[GP1:90,1] + 3.310;
   1:  PR[GP1:91,2] = PR[GP1:90,2] + -28.422;
   1:L PR[91] R[100]mm/sec CNT100;
   1:  PR[GP1:91,1] = PR[GP1:90,1] + 7.343;
   1:  PR[GP1:91,2] = PR[GP1:90,2] + -31.352;
   1:L PR[91] R[100]mm/sec CNT100;
   1:  PR[GP1:91,1] = PR[GP1:90,1] + 10.123;
   1:  PR[GP1:91,2] = PR[GP1:90,2] + -32.803;
   1:L PR[91] R[100]mm/sec CNT100;
   1:  PR[GP1:91,1] = PR[GP1:90,1] + 13.583;
   1:  PR[GP1:91,2] = PR[GP1:90,2] + -33.915;
   1:L PR[91] R[100]mm/sec CNT100;
   1:  PR[GP1:91,1] = PR[GP1:90,1] + 20.029;
   1:  PR[GP1:91,2] = PR[GP1:90,2] + -36.146;
   1:L PR[91] R[100]mm/sec CNT100;
   1:  PR[GP1:91,1] = PR[GP1:90,1] + 23.887;
   1:  PR[GP1:91,2] = PR[GP1:90,2] + -36.654;
   1:L PR[91] R[100]mm/sec CNT100;
   1:  PR[GP1:91,1] = PR[GP1:90,1] + 28.404;
   1:  PR[GP1:91,2] = PR[GP1:90,2] + -36.502;
   1:L PR[91] R[100]mm/sec CNT100;
   1:  PR[GP1:91,1] = PR[GP1:90,1] + 33.735;
   1:  PR[GP1:91,2] = PR[GP1:90,2] + -36.478;
   1:L PR[91] R[100]mm/sec CNT100;
   1:  PR[GP1:91,1] = PR[GP1:90,1] + 38.327;
   1:  PR[GP1:91,2] = PR[GP1:90,2] + -35.490;
   1:L PR[91] R[100]mm/sec CNT100;
   1:  PR[GP1:91,1] = PR[GP1:90,1] + 43.376;
   1:  PR[GP1:91,2] = PR[GP1:90,2] + -33.501;
   1:L PR[91] R[100]mm/sec CNT100;
   1:  PR[GP1:91,1] = PR[GP1:90,1] + 46.776;
   1:  PR[GP1:91,2] = PR[GP1:90,2] + -32.296;
   1:L PR[91] R[100]mm/sec CNT100;
   1:  PR[GP1:91,1] = PR[GP1:90,1] + 51.389;
   1:  PR[GP1:91,2] = PR[GP1:90,2] + -29.436;
   1:L PR[91] R[100]mm/sec CNT100;
   1:  PR[GP1:91,1] = PR[GP1:90,1] + 55.874;
   1:  PR[GP1:91,2] = PR[GP1:90,2] + -25.465;
   1:L PR[91] R[100]mm/sec CNT100;
   1:  PR[GP1:91,1] = PR[GP1:90,1] + 57.462;
   1:  PR[GP1:91,2] = PR[GP1:90,2] + -24.180;
   1:L PR[91] R[100]mm/sec CNT100;
   1:  PR[GP1:91,1] = PR[GP1:90,1] + 61.114;
   1:  PR[GP1:91,2] = PR[GP1:90,2] + -19.438;
   1:L PR[91] R[100]mm/sec CNT100;
   1:  PR[GP1:91,1] = PR[GP1:90,1] + 64.157;
   1:  PR[GP1:91,2] = PR[GP1:90,2] + -13.599;
   1:L PR[91] R[100]mm/sec CNT100;
   1:  PR[GP1:91,1] = PR[GP1:90,1] + 64.647;
   1:  PR[GP1:91,2] = PR[GP1:90,2] + -12.782;
   1:L PR[91] R[100]mm/sec CNT100;
   1:  PR[GP1:91,1] = PR[GP1:90,1] + 66.374;
   1:  PR[GP1:91,2] = PR[GP1:90,2] + -7.004;
   1:L PR[91] R[100]mm/sec CNT100;
   1:  PR[GP1:91,1] = PR[GP1:90,1] + 66.972;
   1:  PR[GP1:91,2] = PR[GP1:90,2] + -0.608;
   1:L PR[91] R[100]mm/sec CNT100;
   1:  PR[GP1:91,1] = PR[GP1:90,1] + 67.075;
   1:  PR[GP1:91,2] = PR[GP1:90,2] + -0.045;
   1:L PR[91] R[100]mm/sec CNT100;
   1:  PR[GP1:91,1] = PR[GP1:90,1] + 66.499;
   1:  PR[GP1:91,2] = PR[GP1:90,2] + 6.202;
   1:L PR[91] R[100]mm/sec CNT100;
   1:  PR[GP1:91,1] = PR[GP1:90,1] + 66.382;
   1:  PR[GP1:91,2] = PR[GP1:90,2] + 6.833;
   1:L PR[91] R[100]mm/sec CNT100;
   1:  PR[GP1:91,1] = PR[GP1:90,1] + 64.642;
   1:  PR[GP1:91,2] = PR[GP1:90,2] + 12.657;
   1:L PR[91] R[100]mm/sec CNT100;
   1:  PR[GP1:91,1] = PR[GP1:90,1] + 61.816;
   1:  PR[GP1:91,2] = PR[GP1:90,2] + 18.133;
   1:L PR[91] R[100]mm/sec CNT100;
   1:  PR[GP1:91,1] = PR[GP1:90,1] + 61.126;
   1:  PR[GP1:91,2] = PR[GP1:90,2] + 19.278;
   1:L PR[91] R[100]mm/sec CNT100;
   1:  PR[GP1:91,1] = PR[GP1:90,1] + 57.453;
   1:  PR[GP1:91,2] = PR[GP1:90,2] + 24.047;
   1:L PR[91] R[100]mm/sec CNT100;
   1:  PR[GP1:91,1] = PR[GP1:90,1] + 53.392;
   1:  PR[GP1:91,2] = PR[GP1:90,2] + 27.679;
   1:L PR[91] R[100]mm/sec CNT100;
   1:  PR[GP1:91,1] = PR[GP1:90,1] + 51.403;
   1:  PR[GP1:91,2] = PR[GP1:90,2] + 29.284;
   1:L PR[91] R[100]mm/sec CNT100;
   1:  PR[GP1:91,1] = PR[GP1:90,1] + 46.768;
   1:  PR[GP1:91,2] = PR[GP1:90,2] + 32.157;
   1:L PR[91] R[100]mm/sec CNT100;
   1:  PR[GP1:91,1] = PR[GP1:90,1] + 42.204;
   1:  PR[GP1:91,2] = PR[GP1:90,2] + 33.980;
   1:L PR[91] R[100]mm/sec CNT100;
   1:  PR[GP1:91,1] = PR[GP1:90,1] + 38.343;
   1:  PR[GP1:91,2] = PR[GP1:90,2] + 35.343;
   1:L PR[91] R[100]mm/sec CNT100;
   1:  PR[GP1:91,1] = PR[GP1:90,1] + 33.731;
   1:  PR[GP1:91,2] = PR[GP1:90,2] + 36.335;
   1:L PR[91] R[100]mm/sec CNT100;
   1:  PR[GP1:91,1] = PR[GP1:90,1] + 29.566;
   1:  PR[GP1:91,2] = PR[GP1:90,2] + 36.492;
   1:L PR[91] R[100]mm/sec CNT100;
   1:  PR[GP1:91,1] = PR[GP1:90,1] + 23.905;
   1:  PR[GP1:91,2] = PR[GP1:90,2] + 36.512;
   1:L PR[91] R[100]mm/sec CNT100;
   1:  PR[GP1:91,1] = PR[GP1:90,1] + 20.031;
   1:  PR[GP1:91,2] = PR[GP1:90,2] + 36.003;
   1:L PR[91] R[100]mm/sec CNT100;
   1:  PR[GP1:91,1] = PR[GP1:90,1] + 16.703;
   1:  PR[GP1:91,2] = PR[GP1:90,2] + 34.944;
   1:L PR[91] R[100]mm/sec CNT100;
   1:  PR[GP1:91,1] = PR[GP1:90,1] + 10.140;
   1:  PR[GP1:91,2] = PR[GP1:90,2] + 32.669;
   1:L PR[91] R[100]mm/sec CNT100;
   1:  PR[GP1:91,1] = PR[GP1:90,1] + 7.346;
   1:  PR[GP1:91,2] = PR[GP1:90,2] + 31.210;
   1:L PR[91] R[100]mm/sec CNT100;
   1:  PR[GP1:91,1] = PR[GP1:90,1] + 4.219;
   1:  PR[GP1:91,2] = PR[GP1:90,2] + 29.002;
   1:L PR[91] R[100]mm/sec CNT100;
   1:  PR[GP1:91,1] = PR[GP1:90,1] + 3.782;
   1:  PR[GP1:91,2] = PR[GP1:90,2] + 28.660;
   1:L PR[91] R[100]mm/sec CNT100;
   1:  PR[GP1:91,1] = PR[GP1:90,1] + 3.357;
   1:  PR[GP1:91,2] = PR[GP1:90,2] + 28.165;
   1:L PR[91] R[100]mm/sec CNT100;
   1:  PR[GP1:91,1] = PR[GP1:90,1] + 1.893;
   1:  PR[GP1:91,2] = PR[GP1:90,2] + 27.587;
   1:L PR[91] R[100]mm/sec CNT100;
   1:  PR[GP1:91,1] = PR[GP1:90,1] + 1.429;
   1:  PR[GP1:91,2] = PR[GP1:90,2] + 27.329;
   1:L PR[91] R[100]mm/sec CNT100;
   1:  ! -- Layer/Ebene 92 -- !;
   1:  PR[91] = PR[90];
   1:  PR[GP1:91,1] = PR[GP1:90,1] + 0.905;
   1:  PR[GP1:91,2] = PR[GP1:90,2] + 27.618;
   1:  PR[GP1:91,3] = PR[GP1:90,3] + 56.425;
   1:L PR[91] R[100]mm/sec CNT100;
   1:  PR[GP1:91,1] = PR[GP1:90,1] + -0.795;
   1:  PR[GP1:91,2] = PR[GP1:90,2] + 28.013;
   1:L PR[91] R[100]mm/sec CNT100;
   1:  PR[GP1:91,1] = PR[GP1:90,1] + -2.719;
   1:  PR[GP1:91,2] = PR[GP1:90,2] + 28.260;
   1:L PR[91] R[100]mm/sec CNT100;
   1:  PR[GP1:91,1] = PR[GP1:90,1] + -3.138;
   1:  PR[GP1:91,2] = PR[GP1:90,2] + 28.473;
   1:L PR[91] R[100]mm/sec CNT100;
   1:  PR[GP1:91,1] = PR[GP1:90,1] + -3.413;
   1:  PR[GP1:91,2] = PR[GP1:90,2] + 28.793;
   1:L PR[91] R[100]mm/sec CNT100;
   1:  PR[GP1:91,1] = PR[GP1:90,1] + -3.680;
   1:  PR[GP1:91,2] = PR[GP1:90,2] + 29.002;
   1:L PR[91] R[100]mm/sec CNT100;
   1:  PR[GP1:91,1] = PR[GP1:90,1] + -6.917;
   1:  PR[GP1:91,2] = PR[GP1:90,2] + 31.289;
   1:L PR[91] R[100]mm/sec CNT100;
   1:  PR[GP1:91,1] = PR[GP1:90,1] + -9.591;
   1:  PR[GP1:91,2] = PR[GP1:90,2] + 32.688;
   1:L PR[91] R[100]mm/sec CNT100;
   1:  PR[GP1:91,1] = PR[GP1:90,1] + -12.892;
   1:  PR[GP1:91,2] = PR[GP1:90,2] + 33.749;
   1:L PR[91] R[100]mm/sec CNT100;
   1:  PR[GP1:91,1] = PR[GP1:90,1] + -19.631;
   1:  PR[GP1:91,2] = PR[GP1:90,2] + 36.079;
   1:L PR[91] R[100]mm/sec CNT100;
   1:  PR[GP1:91,1] = PR[GP1:90,1] + -23.342;
   1:  PR[GP1:91,2] = PR[GP1:90,2] + 36.564;
   1:L PR[91] R[100]mm/sec CNT100;
   1:  PR[GP1:91,1] = PR[GP1:90,1] + -27.704;
   1:  PR[GP1:91,2] = PR[GP1:90,2] + 36.414;
   1:L PR[91] R[100]mm/sec CNT100;
   1:  PR[GP1:91,1] = PR[GP1:90,1] + -33.369;
   1:  PR[GP1:91,2] = PR[GP1:90,2] + 36.385;
   1:L PR[91] R[100]mm/sec CNT100;
   1:  PR[GP1:91,1] = PR[GP1:90,1] + -37.811;
   1:  PR[GP1:91,2] = PR[GP1:90,2] + 35.427;
   1:L PR[91] R[100]mm/sec CNT100;
   1:  PR[GP1:91,1] = PR[GP1:90,1] + -42.682;
   1:  PR[GP1:91,2] = PR[GP1:90,2] + 33.498;
   1:L PR[91] R[100]mm/sec CNT100;
   1:  PR[GP1:91,1] = PR[GP1:90,1] + -46.409;
   1:  PR[GP1:91,2] = PR[GP1:90,2] + 32.175;
   1:L PR[91] R[100]mm/sec CNT100;
   1:  PR[GP1:91,1] = PR[GP1:90,1] + -50.909;
   1:  PR[GP1:91,2] = PR[GP1:90,2] + 29.372;
   1:L PR[91] R[100]mm/sec CNT100;
   1:  PR[GP1:91,1] = PR[GP1:90,1] + -55.283;
   1:  PR[GP1:91,2] = PR[GP1:90,2] + 25.488;
   1:L PR[91] R[100]mm/sec CNT100;
   1:  PR[GP1:91,1] = PR[GP1:90,1] + -57.139;
   1:  PR[GP1:91,2] = PR[GP1:90,2] + 23.986;
   1:L PR[91] R[100]mm/sec CNT100;
   1:  PR[GP1:91,1] = PR[GP1:90,1] + -60.653;
   1:  PR[GP1:91,2] = PR[GP1:90,2] + 19.411;
   1:L PR[91] R[100]mm/sec CNT100;
   1:  PR[GP1:91,1] = PR[GP1:90,1] + -63.603;
   1:  PR[GP1:91,2] = PR[GP1:90,2] + 13.687;
   1:L PR[91] R[100]mm/sec CNT100;
   1:  PR[GP1:91,1] = PR[GP1:90,1] + -64.273;
   1:  PR[GP1:91,2] = PR[GP1:90,2] + 12.569;
   1:L PR[91] R[100]mm/sec CNT100;
   1:  PR[GP1:91,1] = PR[GP1:90,1] + -65.956;
   1:  PR[GP1:91,2] = PR[GP1:90,2] + 6.859;
   1:L PR[91] R[100]mm/sec CNT100;
   1:  PR[GP1:91,1] = PR[GP1:90,1] + -66.510;
   1:  PR[GP1:91,2] = PR[GP1:90,2] + 0.798;
   1:L PR[91] R[100]mm/sec CNT100;
   1:  PR[GP1:91,1] = PR[GP1:90,1] + -66.676;
   1:  PR[GP1:91,2] = PR[GP1:90,2] + -0.100;
   1:L PR[91] R[100]mm/sec CNT100;
   1:  PR[GP1:91,1] = PR[GP1:90,1] + -66.141;
   1:  PR[GP1:91,2] = PR[GP1:90,2] + -6.021;
   1:L PR[91] R[100]mm/sec CNT100;
   1:  PR[GP1:91,1] = PR[GP1:90,1] + -65.963;
   1:  PR[GP1:91,2] = PR[GP1:90,2] + -6.977;
   1:L PR[91] R[100]mm/sec CNT100;
   1:  PR[GP1:91,1] = PR[GP1:90,1] + -64.267;
   1:  PR[GP1:91,2] = PR[GP1:90,2] + -12.733;
   1:L PR[91] R[100]mm/sec CNT100;
   1:  PR[GP1:91,1] = PR[GP1:90,1] + -61.523;
   1:  PR[GP1:91,2] = PR[GP1:90,2] + -18.112;
   1:L PR[91] R[100]mm/sec CNT100;
   1:  PR[GP1:91,1] = PR[GP1:90,1] + -60.665;
   1:  PR[GP1:91,2] = PR[GP1:90,2] + -19.541;
   1:L PR[91] R[100]mm/sec CNT100;
   1:  PR[GP1:91,1] = PR[GP1:90,1] + -57.129;
   1:  PR[GP1:91,2] = PR[GP1:90,2] + -24.143;
   1:L PR[91] R[100]mm/sec CNT100;
   1:  PR[GP1:91,1] = PR[GP1:90,1] + -53.159;
   1:  PR[GP1:91,2] = PR[GP1:90,2] + -27.704;
   1:L PR[91] R[100]mm/sec CNT100;
   1:  PR[GP1:91,1] = PR[GP1:90,1] + -50.919;
   1:  PR[GP1:91,2] = PR[GP1:90,2] + -29.510;
   1:L PR[91] R[100]mm/sec CNT100;
   1:  PR[GP1:91,1] = PR[GP1:90,1] + -46.395;
   1:  PR[GP1:91,2] = PR[GP1:90,2] + -32.328;
   1:L PR[91] R[100]mm/sec CNT100;
   1:  PR[GP1:91,1] = PR[GP1:90,1] + -41.975;
   1:  PR[GP1:91,2] = PR[GP1:90,2] + -34.103;
   1:L PR[91] R[100]mm/sec CNT100;
   1:  PR[GP1:91,1] = PR[GP1:90,1] + -37.816;
   1:  PR[GP1:91,2] = PR[GP1:90,2] + -35.570;
   1:L PR[91] R[100]mm/sec CNT100;
   1:  PR[GP1:91,1] = PR[GP1:90,1] + -33.353;
   1:  PR[GP1:91,2] = PR[GP1:90,2] + -36.533;
   1:L PR[91] R[100]mm/sec CNT100;
   1:  PR[GP1:91,1] = PR[GP1:90,1] + -29.310;
   1:  PR[GP1:91,2] = PR[GP1:90,2] + -36.688;
   1:L PR[91] R[100]mm/sec CNT100;
   1:  PR[GP1:91,1] = PR[GP1:90,1] + -23.341;
   1:  PR[GP1:91,2] = PR[GP1:90,2] + -36.707;
   1:L PR[91] R[100]mm/sec CNT100;
   1:  PR[GP1:91,1] = PR[GP1:90,1] + -19.613;
   1:  PR[GP1:91,2] = PR[GP1:90,2] + -36.220;
   1:L PR[91] R[100]mm/sec CNT100;
   1:  PR[GP1:91,1] = PR[GP1:90,1] + -16.420;
   1:  PR[GP1:91,2] = PR[GP1:90,2] + -35.204;
   1:L PR[91] R[100]mm/sec CNT100;
   1:  PR[GP1:91,1] = PR[GP1:90,1] + -9.586;
   1:  PR[GP1:91,2] = PR[GP1:90,2] + -32.829;
   1:L PR[91] R[100]mm/sec CNT100;
   1:  PR[GP1:91,1] = PR[GP1:90,1] + -6.913;
   1:  PR[GP1:91,2] = PR[GP1:90,2] + -31.431;
   1:L PR[91] R[100]mm/sec CNT100;
   1:  PR[GP1:91,1] = PR[GP1:90,1] + -2.966;
   1:  PR[GP1:91,2] = PR[GP1:90,2] + -28.563;
   1:L PR[91] R[100]mm/sec CNT100;
   1:  PR[GP1:91,1] = PR[GP1:90,1] + -2.568;
   1:  PR[GP1:91,2] = PR[GP1:90,2] + -28.547;
   1:L PR[91] R[100]mm/sec CNT100;
   1:  PR[GP1:91,1] = PR[GP1:90,1] + 1.409;
   1:  PR[GP1:91,2] = PR[GP1:90,2] + -27.698;
   1:L PR[91] R[100]mm/sec CNT100;
   1:  PR[GP1:91,1] = PR[GP1:90,1] + 3.282;
   1:  PR[GP1:91,2] = PR[GP1:90,2] + -28.643;
   1:L PR[91] R[100]mm/sec CNT100;
   1:  PR[GP1:91,1] = PR[GP1:90,1] + 7.131;
   1:  PR[GP1:91,2] = PR[GP1:90,2] + -31.439;
   1:L PR[91] R[100]mm/sec CNT100;
   1:  PR[GP1:91,1] = PR[GP1:90,1] + 9.781;
   1:  PR[GP1:91,2] = PR[GP1:90,2] + -32.822;
   1:L PR[91] R[100]mm/sec CNT100;
   1:  PR[GP1:91,1] = PR[GP1:90,1] + 13.081;
   1:  PR[GP1:91,2] = PR[GP1:90,2] + -33.882;
   1:L PR[91] R[100]mm/sec CNT100;
   1:  PR[GP1:91,1] = PR[GP1:90,1] + 19.830;
   1:  PR[GP1:91,2] = PR[GP1:90,2] + -36.219;
   1:L PR[91] R[100]mm/sec CNT100;
   1:  PR[GP1:91,1] = PR[GP1:90,1] + 23.535;
   1:  PR[GP1:91,2] = PR[GP1:90,2] + -36.706;
   1:L PR[91] R[100]mm/sec CNT100;
   1:  PR[GP1:91,1] = PR[GP1:90,1] + 27.877;
   1:  PR[GP1:91,2] = PR[GP1:90,2] + -36.560;
   1:L PR[91] R[100]mm/sec CNT100;
   1:  PR[GP1:91,1] = PR[GP1:90,1] + 33.548;
   1:  PR[GP1:91,2] = PR[GP1:90,2] + -36.535;
   1:L PR[91] R[100]mm/sec CNT100;
   1:  PR[GP1:91,1] = PR[GP1:90,1] + 37.982;
   1:  PR[GP1:91,2] = PR[GP1:90,2] + -35.580;
   1:L PR[91] R[100]mm/sec CNT100;
   1:  PR[GP1:91,1] = PR[GP1:90,1] + 42.861;
   1:  PR[GP1:91,2] = PR[GP1:90,2] + -33.658;
   1:L PR[91] R[100]mm/sec CNT100;
   1:  PR[GP1:91,1] = PR[GP1:90,1] + 46.593;
   1:  PR[GP1:91,2] = PR[GP1:90,2] + -32.336;
   1:L PR[91] R[100]mm/sec CNT100;
   1:  PR[GP1:91,1] = PR[GP1:90,1] + 51.065;
   1:  PR[GP1:91,2] = PR[GP1:90,2] + -29.563;
   1:L PR[91] R[100]mm/sec CNT100;
   1:  PR[GP1:91,1] = PR[GP1:90,1] + 55.416;
   1:  PR[GP1:91,2] = PR[GP1:90,2] + -25.711;
   1:L PR[91] R[100]mm/sec CNT100;
   1:  PR[GP1:91,1] = PR[GP1:90,1] + 57.280;
   1:  PR[GP1:91,2] = PR[GP1:90,2] + -24.202;
   1:L PR[91] R[100]mm/sec CNT100;
   1:  PR[GP1:91,1] = PR[GP1:90,1] + 60.831;
   1:  PR[GP1:91,2] = PR[GP1:90,2] + -19.593;
   1:L PR[91] R[100]mm/sec CNT100;
   1:  PR[GP1:91,1] = PR[GP1:90,1] + 63.790;
   1:  PR[GP1:91,2] = PR[GP1:90,2] + -13.915;
   1:L PR[91] R[100]mm/sec CNT100;
   1:  PR[GP1:91,1] = PR[GP1:90,1] + 64.461;
   1:  PR[GP1:91,2] = PR[GP1:90,2] + -12.796;
   1:L PR[91] R[100]mm/sec CNT100;
   1:  PR[GP1:91,1] = PR[GP1:90,1] + 66.142;
   1:  PR[GP1:91,2] = PR[GP1:90,2] + -7.171;
   1:L PR[91] R[100]mm/sec CNT100;
   1:  PR[GP1:91,1] = PR[GP1:90,1] + 66.724;
   1:  PR[GP1:91,2] = PR[GP1:90,2] + -0.943;
   1:L PR[91] R[100]mm/sec CNT100;
   1:  PR[GP1:91,1] = PR[GP1:90,1] + 66.889;
   1:  PR[GP1:91,2] = PR[GP1:90,2] + -0.045;
   1:L PR[91] R[100]mm/sec CNT100;
   1:  PR[GP1:91,1] = PR[GP1:90,1] + 66.327;
   1:  PR[GP1:91,2] = PR[GP1:90,2] + 6.041;
   1:L PR[91] R[100]mm/sec CNT100;
   1:  PR[GP1:91,1] = PR[GP1:90,1] + 66.149;
   1:  PR[GP1:91,2] = PR[GP1:90,2] + 7.001;
   1:L PR[91] R[100]mm/sec CNT100;
   1:  PR[GP1:91,1] = PR[GP1:90,1] + 64.456;
   1:  PR[GP1:91,2] = PR[GP1:90,2] + 12.670;
   1:L PR[91] R[100]mm/sec CNT100;
   1:  PR[GP1:91,1] = PR[GP1:90,1] + 61.704;
   1:  PR[GP1:91,2] = PR[GP1:90,2] + 18.003;
   1:L PR[91] R[100]mm/sec CNT100;
   1:  PR[GP1:91,1] = PR[GP1:90,1] + 60.843;
   1:  PR[GP1:91,2] = PR[GP1:90,2] + 19.433;
   1:L PR[91] R[100]mm/sec CNT100;
   1:  PR[GP1:91,1] = PR[GP1:90,1] + 57.272;
   1:  PR[GP1:91,2] = PR[GP1:90,2] + 24.069;
   1:L PR[91] R[100]mm/sec CNT100;
   1:  PR[GP1:91,1] = PR[GP1:90,1] + 53.323;
   1:  PR[GP1:91,2] = PR[GP1:90,2] + 27.600;
   1:L PR[91] R[100]mm/sec CNT100;
   1:  PR[GP1:91,1] = PR[GP1:90,1] + 51.080;
   1:  PR[GP1:91,2] = PR[GP1:90,2] + 29.411;
   1:L PR[91] R[100]mm/sec CNT100;
   1:  PR[GP1:91,1] = PR[GP1:90,1] + 46.586;
   1:  PR[GP1:91,2] = PR[GP1:90,2] + 32.196;
   1:L PR[91] R[100]mm/sec CNT100;
   1:  PR[GP1:91,1] = PR[GP1:90,1] + 42.159;
   1:  PR[GP1:91,2] = PR[GP1:90,2] + 33.964;
   1:L PR[91] R[100]mm/sec CNT100;
   1:  PR[GP1:91,1] = PR[GP1:90,1] + 37.999;
   1:  PR[GP1:91,2] = PR[GP1:90,2] + 35.433;
   1:L PR[91] R[100]mm/sec CNT100;
   1:  PR[GP1:91,1] = PR[GP1:90,1] + 33.544;
   1:  PR[GP1:91,2] = PR[GP1:90,2] + 36.392;
   1:L PR[91] R[100]mm/sec CNT100;
   1:  PR[GP1:91,1] = PR[GP1:90,1] + 29.521;
   1:  PR[GP1:91,2] = PR[GP1:90,2] + 36.544;
   1:L PR[91] R[100]mm/sec CNT100;
   1:  PR[GP1:91,1] = PR[GP1:90,1] + 23.554;
   1:  PR[GP1:91,2] = PR[GP1:90,2] + 36.565;
   1:L PR[91] R[100]mm/sec CNT100;
   1:  PR[GP1:91,1] = PR[GP1:90,1] + 19.833;
   1:  PR[GP1:91,2] = PR[GP1:90,2] + 36.075;
   1:L PR[91] R[100]mm/sec CNT100;
   1:  PR[GP1:91,1] = PR[GP1:90,1] + 16.635;
   1:  PR[GP1:91,2] = PR[GP1:90,2] + 35.058;
   1:L PR[91] R[100]mm/sec CNT100;
   1:  PR[GP1:91,1] = PR[GP1:90,1] + 9.798;
   1:  PR[GP1:91,2] = PR[GP1:90,2] + 32.688;
   1:L PR[91] R[100]mm/sec CNT100;
   1:  PR[GP1:91,1] = PR[GP1:90,1] + 7.134;
   1:  PR[GP1:91,2] = PR[GP1:90,2] + 31.297;
   1:L PR[91] R[100]mm/sec CNT100;
   1:  PR[GP1:91,1] = PR[GP1:90,1] + 3.889;
   1:  PR[GP1:91,2] = PR[GP1:90,2] + 29.005;
   1:L PR[91] R[100]mm/sec CNT100;
   1:  PR[GP1:91,1] = PR[GP1:90,1] + 3.624;
   1:  PR[GP1:91,2] = PR[GP1:90,2] + 28.797;
   1:L PR[91] R[100]mm/sec CNT100;
   1:  PR[GP1:91,1] = PR[GP1:90,1] + 3.327;
   1:  PR[GP1:91,2] = PR[GP1:90,2] + 28.452;
   1:L PR[91] R[100]mm/sec CNT100;
   1:  PR[GP1:91,1] = PR[GP1:90,1] + 2.338;
   1:  PR[GP1:91,2] = PR[GP1:90,2] + 28.061;
   1:L PR[91] R[100]mm/sec CNT100;
   1:  PR[GP1:91,1] = PR[GP1:90,1] + 1.459;
   1:  PR[GP1:91,2] = PR[GP1:90,2] + 27.572;
   1:L PR[91] R[100]mm/sec CNT100;
   1:  ! -- Layer/Ebene 93 -- !;
   1:  PR[91] = PR[90];
   1:  PR[GP1:91,1] = PR[GP1:90,1] + 0.755;
   1:  PR[GP1:91,2] = PR[GP1:90,2] + 27.876;
   1:  PR[GP1:91,3] = PR[GP1:90,3] + 57.035;
   1:L PR[91] R[100]mm/sec CNT100;
   1:  PR[GP1:91,1] = PR[GP1:90,1] + -1.875;
   1:  PR[GP1:91,2] = PR[GP1:90,2] + 28.487;
   1:L PR[91] R[100]mm/sec CNT100;
   1:  PR[GP1:91,1] = PR[GP1:90,1] + -2.808;
   1:  PR[GP1:91,2] = PR[GP1:90,2] + 28.607;
   1:L PR[91] R[100]mm/sec CNT100;
   1:  PR[GP1:91,1] = PR[GP1:90,1] + -3.109;
   1:  PR[GP1:91,2] = PR[GP1:90,2] + 28.760;
   1:L PR[91] R[100]mm/sec CNT100;
   1:  PR[GP1:91,1] = PR[GP1:90,1] + -3.257;
   1:  PR[GP1:91,2] = PR[GP1:90,2] + 28.933;
   1:L PR[91] R[100]mm/sec CNT100;
   1:  PR[GP1:91,1] = PR[GP1:90,1] + -3.350;
   1:  PR[GP1:91,2] = PR[GP1:90,2] + 29.005;
   1:L PR[91] R[100]mm/sec CNT100;
   1:  PR[GP1:91,1] = PR[GP1:90,1] + -6.706;
   1:  PR[GP1:91,2] = PR[GP1:90,2] + 31.377;
   1:L PR[91] R[100]mm/sec CNT100;
   1:  PR[GP1:91,1] = PR[GP1:90,1] + -9.249;
   1:  PR[GP1:91,2] = PR[GP1:90,2] + 32.707;
   1:L PR[91] R[100]mm/sec CNT100;
   1:  PR[GP1:91,1] = PR[GP1:90,1] + -12.391;
   1:  PR[GP1:91,2] = PR[GP1:90,2] + 33.717;
   1:L PR[91] R[100]mm/sec CNT100;
   1:  PR[GP1:91,1] = PR[GP1:90,1] + -19.433;
   1:  PR[GP1:91,2] = PR[GP1:90,2] + 36.151;
   1:L PR[91] R[100]mm/sec CNT100;
   1:  PR[GP1:91,1] = PR[GP1:90,1] + -22.990;
   1:  PR[GP1:91,2] = PR[GP1:90,2] + 36.616;
   1:L PR[91] R[100]mm/sec CNT100;
   1:  PR[GP1:91,1] = PR[GP1:90,1] + -27.176;
   1:  PR[GP1:91,2] = PR[GP1:90,2] + 36.472;
   1:L PR[91] R[100]mm/sec CNT100;
   1:  PR[GP1:91,1] = PR[GP1:90,1] + -33.181;
   1:  PR[GP1:91,2] = PR[GP1:90,2] + 36.442;
   1:L PR[91] R[100]mm/sec CNT100;
   1:  PR[GP1:91,1] = PR[GP1:90,1] + -37.465;
   1:  PR[GP1:91,2] = PR[GP1:90,2] + 35.518;
   1:L PR[91] R[100]mm/sec CNT100;
   1:  PR[GP1:91,1] = PR[GP1:90,1] + -42.167;
   1:  PR[GP1:91,2] = PR[GP1:90,2] + 33.656;
   1:L PR[91] R[100]mm/sec CNT100;
   1:  PR[GP1:91,1] = PR[GP1:90,1] + -46.225;
   1:  PR[GP1:91,2] = PR[GP1:90,2] + 32.215;
   1:L PR[91] R[100]mm/sec CNT100;
   1:  PR[GP1:91,1] = PR[GP1:90,1] + -50.584;
   1:  PR[GP1:91,2] = PR[GP1:90,2] + 29.500;
   1:L PR[91] R[100]mm/sec CNT100;
   1:  PR[GP1:91,1] = PR[GP1:90,1] + -54.823;
   1:  PR[GP1:91,2] = PR[GP1:90,2] + 25.736;
   1:L PR[91] R[100]mm/sec CNT100;
   1:  PR[GP1:91,1] = PR[GP1:90,1] + -56.956;
   1:  PR[GP1:91,2] = PR[GP1:90,2] + 24.010;
   1:L PR[91] R[100]mm/sec CNT100;
   1:  PR[GP1:91,1] = PR[GP1:90,1] + -60.369;
   1:  PR[GP1:91,2] = PR[GP1:90,2] + 19.567;
   1:L PR[91] R[100]mm/sec CNT100;
   1:  PR[GP1:91,1] = PR[GP1:90,1] + -63.235;
   1:  PR[GP1:91,2] = PR[GP1:90,2] + 14.005;
   1:L PR[91] R[100]mm/sec CNT100;
   1:  PR[GP1:91,1] = PR[GP1:90,1] + -64.086;
   1:  PR[GP1:91,2] = PR[GP1:90,2] + 12.584;
   1:L PR[91] R[100]mm/sec CNT100;
   1:  PR[GP1:91,1] = PR[GP1:90,1] + -65.723;
   1:  PR[GP1:91,2] = PR[GP1:90,2] + 7.031;
   1:L PR[91] R[100]mm/sec CNT100;
   1:  PR[GP1:91,1] = PR[GP1:90,1] + -66.262;
   1:  PR[GP1:91,2] = PR[GP1:90,2] + 1.132;
   1:L PR[91] R[100]mm/sec CNT100;
   1:  PR[GP1:91,1] = PR[GP1:90,1] + -66.490;
   1:  PR[GP1:91,2] = PR[GP1:90,2] + -0.100;
   1:L PR[91] R[100]mm/sec CNT100;
   1:  PR[GP1:91,1] = PR[GP1:90,1] + -65.969;
   1:  PR[GP1:91,2] = PR[GP1:90,2] + -5.865;
   1:L PR[91] R[100]mm/sec CNT100;
   1:  PR[GP1:91,1] = PR[GP1:90,1] + -65.730;
   1:  PR[GP1:91,2] = PR[GP1:90,2] + -7.149;
   1:L PR[91] R[100]mm/sec CNT100;
   1:  PR[GP1:91,1] = PR[GP1:90,1] + -64.080;
   1:  PR[GP1:91,2] = PR[GP1:90,2] + -12.749;
   1:L PR[91] R[100]mm/sec CNT100;
   1:  PR[GP1:91,1] = PR[GP1:90,1] + -61.410;
   1:  PR[GP1:91,2] = PR[GP1:90,2] + -17.982;
   1:L PR[91] R[100]mm/sec CNT100;
   1:  PR[GP1:91,1] = PR[GP1:90,1] + -60.380;
   1:  PR[GP1:91,2] = PR[GP1:90,2] + -19.697;
   1:L PR[91] R[100]mm/sec CNT100;
   1:  PR[GP1:91,1] = PR[GP1:90,1] + -56.945;
   1:  PR[GP1:91,2] = PR[GP1:90,2] + -24.167;
   1:L PR[91] R[100]mm/sec CNT100;
   1:  PR[GP1:91,1] = PR[GP1:90,1] + -53.088;
   1:  PR[GP1:91,2] = PR[GP1:90,2] + -27.627;
   1:L PR[91] R[100]mm/sec CNT100;
   1:  PR[GP1:91,1] = PR[GP1:90,1] + -50.593;
   1:  PR[GP1:91,2] = PR[GP1:90,2] + -29.638;
   1:L PR[91] R[100]mm/sec CNT100;
   1:  PR[GP1:91,1] = PR[GP1:90,1] + -46.211;
   1:  PR[GP1:91,2] = PR[GP1:90,2] + -32.368;
   1:L PR[91] R[100]mm/sec CNT100;
   1:  PR[GP1:91,1] = PR[GP1:90,1] + -41.929;
   1:  PR[GP1:91,2] = PR[GP1:90,2] + -34.087;
   1:L PR[91] R[100]mm/sec CNT100;
   1:  PR[GP1:91,1] = PR[GP1:90,1] + -37.470;
   1:  PR[GP1:91,2] = PR[GP1:90,2] + -35.661;
   1:L PR[91] R[100]mm/sec CNT100;
   1:  PR[GP1:91,1] = PR[GP1:90,1] + -33.165;
   1:  PR[GP1:91,2] = PR[GP1:90,2] + -36.589;
   1:L PR[91] R[100]mm/sec CNT100;
   1:  PR[GP1:91,1] = PR[GP1:90,1] + -29.264;
   1:  PR[GP1:91,2] = PR[GP1:90,2] + -36.740;
   1:L PR[91] R[100]mm/sec CNT100;
   1:  PR[GP1:91,1] = PR[GP1:90,1] + -22.989;
   1:  PR[GP1:91,2] = PR[GP1:90,2] + -36.759;
   1:L PR[91] R[100]mm/sec CNT100;
   1:  PR[GP1:91,1] = PR[GP1:90,1] + -19.415;
   1:  PR[GP1:91,2] = PR[GP1:90,2] + -36.292;
   1:L PR[91] R[100]mm/sec CNT100;
   1:  PR[GP1:91,1] = PR[GP1:90,1] + -16.352;
   1:  PR[GP1:91,2] = PR[GP1:90,2] + -35.318;
   1:L PR[91] R[100]mm/sec CNT100;
   1:  PR[GP1:91,1] = PR[GP1:90,1] + -9.244;
   1:  PR[GP1:91,2] = PR[GP1:90,2] + -32.848;
   1:L PR[91] R[100]mm/sec CNT100;
   1:  PR[GP1:91,1] = PR[GP1:90,1] + -6.702;
   1:  PR[GP1:91,2] = PR[GP1:90,2] + -31.518;
   1:L PR[91] R[100]mm/sec CNT100;
   1:  PR[GP1:91,1] = PR[GP1:90,1] + -2.938;
   1:  PR[GP1:91,2] = PR[GP1:90,2] + -28.783;
   1:L PR[91] R[100]mm/sec CNT100;
   1:  PR[GP1:91,1] = PR[GP1:90,1] + -2.402;
   1:  PR[GP1:91,2] = PR[GP1:90,2] + -28.762;
   1:L PR[91] R[100]mm/sec CNT100;
   1:  PR[GP1:91,1] = PR[GP1:90,1] + 1.512;
   1:  PR[GP1:91,2] = PR[GP1:90,2] + -27.926;
   1:L PR[91] R[100]mm/sec CNT100;
   1:  PR[GP1:91,1] = PR[GP1:90,1] + 1.735;
   1:  PR[GP1:91,2] = PR[GP1:90,2] + -28.106;
   1:L PR[91] R[100]mm/sec CNT100;
   1:  PR[GP1:91,1] = PR[GP1:90,1] + 3.253;
   1:  PR[GP1:91,2] = PR[GP1:90,2] + -28.862;
   1:L PR[91] R[100]mm/sec CNT100;
   1:  PR[GP1:91,1] = PR[GP1:90,1] + 6.919;
   1:  PR[GP1:91,2] = PR[GP1:90,2] + -31.526;
   1:L PR[91] R[100]mm/sec CNT100;
   1:  PR[GP1:91,1] = PR[GP1:90,1] + 9.439;
   1:  PR[GP1:91,2] = PR[GP1:90,2] + -32.840;
   1:L PR[91] R[100]mm/sec CNT100;
   1:  PR[GP1:91,1] = PR[GP1:90,1] + 12.580;
   1:  PR[GP1:91,2] = PR[GP1:90,2] + -33.849;
   1:L PR[91] R[100]mm/sec CNT100;
   1:  PR[GP1:91,1] = PR[GP1:90,1] + 19.631;
   1:  PR[GP1:91,2] = PR[GP1:90,2] + -36.291;
   1:L PR[91] R[100]mm/sec CNT100;
   1:  PR[GP1:91,1] = PR[GP1:90,1] + 23.183;
   1:  PR[GP1:91,2] = PR[GP1:90,2] + -36.758;
   1:L PR[91] R[100]mm/sec CNT100;
   1:  PR[GP1:91,1] = PR[GP1:90,1] + 27.349;
   1:  PR[GP1:91,2] = PR[GP1:90,2] + -36.618;
   1:L PR[91] R[100]mm/sec CNT100;
   1:  PR[GP1:91,1] = PR[GP1:90,1] + 33.360;
   1:  PR[GP1:91,2] = PR[GP1:90,2] + -36.591;
   1:L PR[91] R[100]mm/sec CNT100;
   1:  PR[GP1:91,1] = PR[GP1:90,1] + 37.638;
   1:  PR[GP1:91,2] = PR[GP1:90,2] + -35.671;
   1:L PR[91] R[100]mm/sec CNT100;
   1:  PR[GP1:91,1] = PR[GP1:90,1] + 42.346;
   1:  PR[GP1:91,2] = PR[GP1:90,2] + -33.816;
   1:L PR[91] R[100]mm/sec CNT100;
   1:  PR[GP1:91,1] = PR[GP1:90,1] + 46.410;
   1:  PR[GP1:91,2] = PR[GP1:90,2] + -32.376;
   1:L PR[91] R[100]mm/sec CNT100;
   1:  PR[GP1:91,1] = PR[GP1:90,1] + 50.742;
   1:  PR[GP1:91,2] = PR[GP1:90,2] + -29.690;
   1:L PR[91] R[100]mm/sec CNT100;
   1:  PR[GP1:91,1] = PR[GP1:90,1] + 54.957;
   1:  PR[GP1:91,2] = PR[GP1:90,2] + -25.958;
   1:L PR[91] R[100]mm/sec CNT100;
   1:  PR[GP1:91,1] = PR[GP1:90,1] + 57.098;
   1:  PR[GP1:91,2] = PR[GP1:90,2] + -24.224;
   1:L PR[91] R[100]mm/sec CNT100;
   1:  PR[GP1:91,1] = PR[GP1:90,1] + 60.547;
   1:  PR[GP1:91,2] = PR[GP1:90,2] + -19.747;
   1:L PR[91] R[100]mm/sec CNT100;
   1:  PR[GP1:91,1] = PR[GP1:90,1] + 63.422;
   1:  PR[GP1:91,2] = PR[GP1:90,2] + -14.231;
   1:L PR[91] R[100]mm/sec CNT100;
   1:  PR[GP1:91,1] = PR[GP1:90,1] + 64.275;
   1:  PR[GP1:91,2] = PR[GP1:90,2] + -12.810;
   1:L PR[91] R[100]mm/sec CNT100;
   1:  PR[GP1:91,1] = PR[GP1:90,1] + 65.909;
   1:  PR[GP1:91,2] = PR[GP1:90,2] + -7.339;
   1:L PR[91] R[100]mm/sec CNT100;
   1:  PR[GP1:91,1] = PR[GP1:90,1] + 66.476;
   1:  PR[GP1:91,2] = PR[GP1:90,2] + -1.278;
   1:L PR[91] R[100]mm/sec CNT100;
   1:  PR[GP1:91,1] = PR[GP1:90,1] + 66.703;
   1:  PR[GP1:91,2] = PR[GP1:90,2] + -0.045;
   1:L PR[91] R[100]mm/sec CNT100;
   1:  PR[GP1:91,1] = PR[GP1:90,1] + 66.156;
   1:  PR[GP1:91,2] = PR[GP1:90,2] + 5.881;
   1:L PR[91] R[100]mm/sec CNT100;
   1:  PR[GP1:91,1] = PR[GP1:90,1] + 65.917;
   1:  PR[GP1:91,2] = PR[GP1:90,2] + 7.169;
   1:L PR[91] R[100]mm/sec CNT100;
   1:  PR[GP1:91,1] = PR[GP1:90,1] + 64.269;
   1:  PR[GP1:91,2] = PR[GP1:90,2] + 12.684;
   1:L PR[91] R[100]mm/sec CNT100;
   1:  PR[GP1:91,1] = PR[GP1:90,1] + 61.592;
   1:  PR[GP1:91,2] = PR[GP1:90,2] + 17.873;
   1:L PR[91] R[100]mm/sec CNT100;
   1:  PR[GP1:91,1] = PR[GP1:90,1] + 60.559;
   1:  PR[GP1:91,2] = PR[GP1:90,2] + 19.588;
   1:L PR[91] R[100]mm/sec CNT100;
   1:  PR[GP1:91,1] = PR[GP1:90,1] + 57.090;
   1:  PR[GP1:91,2] = PR[GP1:90,2] + 24.091;
   1:L PR[91] R[100]mm/sec CNT100;
   1:  PR[GP1:91,1] = PR[GP1:90,1] + 53.254;
   1:  PR[GP1:91,2] = PR[GP1:90,2] + 27.521;
   1:L PR[91] R[100]mm/sec CNT100;
   1:  PR[GP1:91,1] = PR[GP1:90,1] + 50.756;
   1:  PR[GP1:91,2] = PR[GP1:90,2] + 29.538;
   1:L PR[91] R[100]mm/sec CNT100;
   1:  PR[GP1:91,1] = PR[GP1:90,1] + 46.403;
   1:  PR[GP1:91,2] = PR[GP1:90,2] + 32.236;
   1:L PR[91] R[100]mm/sec CNT100;
   1:  PR[GP1:91,1] = PR[GP1:90,1] + 42.115;
   1:  PR[GP1:91,2] = PR[GP1:90,2] + 33.949;
   1:L PR[91] R[100]mm/sec CNT100;
   1:  PR[GP1:91,1] = PR[GP1:90,1] + 37.654;
   1:  PR[GP1:91,2] = PR[GP1:90,2] + 35.523;
   1:L PR[91] R[100]mm/sec CNT100;
   1:  PR[GP1:91,1] = PR[GP1:90,1] + 33.357;
   1:  PR[GP1:91,2] = PR[GP1:90,2] + 36.448;
   1:L PR[91] R[100]mm/sec CNT100;
   1:  PR[GP1:91,1] = PR[GP1:90,1] + 29.476;
   1:  PR[GP1:91,2] = PR[GP1:90,2] + 36.595;
   1:L PR[91] R[100]mm/sec CNT100;
   1:  PR[GP1:91,1] = PR[GP1:90,1] + 23.203;
   1:  PR[GP1:91,2] = PR[GP1:90,2] + 36.617;
   1:L PR[91] R[100]mm/sec CNT100;
   1:  PR[GP1:91,1] = PR[GP1:90,1] + 19.634;
   1:  PR[GP1:91,2] = PR[GP1:90,2] + 36.148;
   1:L PR[91] R[100]mm/sec CNT100;
   1:  PR[GP1:91,1] = PR[GP1:90,1] + 16.567;
   1:  PR[GP1:91,2] = PR[GP1:90,2] + 35.172;
   1:L PR[91] R[100]mm/sec CNT100;
   1:  PR[GP1:91,1] = PR[GP1:90,1] + 9.457;
   1:  PR[GP1:91,2] = PR[GP1:90,2] + 32.706;
   1:L PR[91] R[100]mm/sec CNT100;
   1:  PR[GP1:91,1] = PR[GP1:90,1] + 6.923;
   1:  PR[GP1:91,2] = PR[GP1:90,2] + 31.384;
   1:L PR[91] R[100]mm/sec CNT100;
   1:  PR[GP1:91,1] = PR[GP1:90,1] + 3.558;
   1:  PR[GP1:91,2] = PR[GP1:90,2] + 29.007;
   1:L PR[91] R[100]mm/sec CNT100;
   1:  PR[GP1:91,1] = PR[GP1:90,1] + 3.466;
   1:  PR[GP1:91,2] = PR[GP1:90,2] + 28.935;
   1:L PR[91] R[100]mm/sec CNT100;
   1:  PR[GP1:91,1] = PR[GP1:90,1] + 3.297;
   1:  PR[GP1:91,2] = PR[GP1:90,2] + 28.739;
   1:L PR[91] R[100]mm/sec CNT100;
   1:  PR[GP1:91,1] = PR[GP1:90,1] + 2.783;
   1:  PR[GP1:91,2] = PR[GP1:90,2] + 28.536;
   1:L PR[91] R[100]mm/sec CNT100;
   1:  PR[GP1:91,1] = PR[GP1:90,1] + 1.489;
   1:  PR[GP1:91,2] = PR[GP1:90,2] + 27.816;
   1:L PR[91] R[100]mm/sec CNT100;
   1:  ! -- Layer/Ebene 94 -- !;
   1:  PR[91] = PR[90];
   1:  PR[GP1:91,1] = PR[GP1:90,1] + 0.604;
   1:  PR[GP1:91,2] = PR[GP1:90,2] + 28.134;
   1:  PR[GP1:91,3] = PR[GP1:90,3] + 57.645;
   1:L PR[91] R[100]mm/sec CNT100;
   1:  PR[GP1:91,1] = PR[GP1:90,1] + -2.952;
   1:  PR[GP1:91,2] = PR[GP1:90,2] + 28.961;
   1:L PR[91] R[100]mm/sec CNT100;
   1:  PR[GP1:91,1] = PR[GP1:90,1] + -6.495;
   1:  PR[GP1:91,2] = PR[GP1:90,2] + 31.464;
   1:L PR[91] R[100]mm/sec CNT100;
   1:  PR[GP1:91,1] = PR[GP1:90,1] + -8.907;
   1:  PR[GP1:91,2] = PR[GP1:90,2] + 32.726;
   1:L PR[91] R[100]mm/sec CNT100;
   1:  PR[GP1:91,1] = PR[GP1:90,1] + -11.890;
   1:  PR[GP1:91,2] = PR[GP1:90,2] + 33.684;
   1:L PR[91] R[100]mm/sec CNT100;
   1:  PR[GP1:91,1] = PR[GP1:90,1] + -19.235;
   1:  PR[GP1:91,2] = PR[GP1:90,2] + 36.223;
   1:L PR[91] R[100]mm/sec CNT100;
   1:  PR[GP1:91,1] = PR[GP1:90,1] + -22.639;
   1:  PR[GP1:91,2] = PR[GP1:90,2] + 36.668;
   1:L PR[91] R[100]mm/sec CNT100;
   1:  PR[GP1:91,1] = PR[GP1:90,1] + -26.648;
   1:  PR[GP1:91,2] = PR[GP1:90,2] + 36.530;
   1:L PR[91] R[100]mm/sec CNT100;
   1:  PR[GP1:91,1] = PR[GP1:90,1] + -32.994;
   1:  PR[GP1:91,2] = PR[GP1:90,2] + 36.499;
   1:L PR[91] R[100]mm/sec CNT100;
   1:  PR[GP1:91,1] = PR[GP1:90,1] + -37.119;
   1:  PR[GP1:91,2] = PR[GP1:90,2] + 35.609;
   1:L PR[91] R[100]mm/sec CNT100;
   1:  PR[GP1:91,1] = PR[GP1:90,1] + -41.651;
   1:  PR[GP1:91,2] = PR[GP1:90,2] + 33.814;
   1:L PR[91] R[100]mm/sec CNT100;
   1:  PR[GP1:91,1] = PR[GP1:90,1] + -46.042;
   1:  PR[GP1:91,2] = PR[GP1:90,2] + 32.255;
   1:L PR[91] R[100]mm/sec CNT100;
   1:  PR[GP1:91,1] = PR[GP1:90,1] + -50.259;
   1:  PR[GP1:91,2] = PR[GP1:90,2] + 29.628;
   1:L PR[91] R[100]mm/sec CNT100;
   1:  PR[GP1:91,1] = PR[GP1:90,1] + -54.362;
   1:  PR[GP1:91,2] = PR[GP1:90,2] + 25.984;
   1:L PR[91] R[100]mm/sec CNT100;
   1:  PR[GP1:91,1] = PR[GP1:90,1] + -56.772;
   1:  PR[GP1:91,2] = PR[GP1:90,2] + 24.034;
   1:L PR[91] R[100]mm/sec CNT100;
   1:  PR[GP1:91,1] = PR[GP1:90,1] + -60.084;
   1:  PR[GP1:91,2] = PR[GP1:90,2] + 19.723;
   1:L PR[91] R[100]mm/sec CNT100;
   1:  PR[GP1:91,1] = PR[GP1:90,1] + -62.867;
   1:  PR[GP1:91,2] = PR[GP1:90,2] + 14.323;
   1:L PR[91] R[100]mm/sec CNT100;
   1:  PR[GP1:91,1] = PR[GP1:90,1] + -63.899;
   1:  PR[GP1:91,2] = PR[GP1:90,2] + 12.600;
   1:L PR[91] R[100]mm/sec CNT100;
   1:  PR[GP1:91,1] = PR[GP1:90,1] + -65.490;
   1:  PR[GP1:91,2] = PR[GP1:90,2] + 7.203;
   1:L PR[91] R[100]mm/sec CNT100;
   1:  PR[GP1:91,1] = PR[GP1:90,1] + -66.014;
   1:  PR[GP1:91,2] = PR[GP1:90,2] + 1.467;
   1:L PR[91] R[100]mm/sec CNT100;
   1:  PR[GP1:91,1] = PR[GP1:90,1] + -66.303;
   1:  PR[GP1:91,2] = PR[GP1:90,2] + -0.100;
   1:L PR[91] R[100]mm/sec CNT100;
   1:  PR[GP1:91,1] = PR[GP1:90,1] + -65.797;
   1:  PR[GP1:91,2] = PR[GP1:90,2] + -5.708;
   1:L PR[91] R[100]mm/sec CNT100;
   1:  PR[GP1:91,1] = PR[GP1:90,1] + -65.497;
   1:  PR[GP1:91,2] = PR[GP1:90,2] + -7.320;
   1:L PR[91] R[100]mm/sec CNT100;
   1:  PR[GP1:91,1] = PR[GP1:90,1] + -63.893;
   1:  PR[GP1:91,2] = PR[GP1:90,2] + -12.764;
   1:L PR[91] R[100]mm/sec CNT100;
   1:  PR[GP1:91,1] = PR[GP1:90,1] + -61.298;
   1:  PR[GP1:91,2] = PR[GP1:90,2] + -17.852;
   1:L PR[91] R[100]mm/sec CNT100;
   1:  PR[GP1:91,1] = PR[GP1:90,1] + -60.095;
   1:  PR[GP1:91,2] = PR[GP1:90,2] + -19.853;
   1:L PR[91] R[100]mm/sec CNT100;
   1:  PR[GP1:91,1] = PR[GP1:90,1] + -56.762;
   1:  PR[GP1:91,2] = PR[GP1:90,2] + -24.192;
   1:L PR[91] R[100]mm/sec CNT100;
   1:  PR[GP1:91,1] = PR[GP1:90,1] + -53.018;
   1:  PR[GP1:91,2] = PR[GP1:90,2] + -27.550;
   1:L PR[91] R[100]mm/sec CNT100;
   1:  PR[GP1:91,1] = PR[GP1:90,1] + -50.268;
   1:  PR[GP1:91,2] = PR[GP1:90,2] + -29.766;
   1:L PR[91] R[100]mm/sec CNT100;
   1:  PR[GP1:91,1] = PR[GP1:90,1] + -46.028;
   1:  PR[GP1:91,2] = PR[GP1:90,2] + -32.408;
   1:L PR[91] R[100]mm/sec CNT100;
   1:  PR[GP1:91,1] = PR[GP1:90,1] + -41.883;
   1:  PR[GP1:91,2] = PR[GP1:90,2] + -34.072;
   1:L PR[91] R[100]mm/sec CNT100;
   1:  PR[GP1:91,1] = PR[GP1:90,1] + -37.124;
   1:  PR[GP1:91,2] = PR[GP1:90,2] + -35.751;
   1:L PR[91] R[100]mm/sec CNT100;
   1:  PR[GP1:91,1] = PR[GP1:90,1] + -32.976;
   1:  PR[GP1:91,2] = PR[GP1:90,2] + -36.646;
   1:L PR[91] R[100]mm/sec CNT100;
   1:  PR[GP1:91,1] = PR[GP1:90,1] + -29.218;
   1:  PR[GP1:91,2] = PR[GP1:90,2] + -36.791;
   1:L PR[91] R[100]mm/sec CNT100;
   1:  PR[GP1:91,1] = PR[GP1:90,1] + -22.637;
   1:  PR[GP1:91,2] = PR[GP1:90,2] + -36.812;
   1:L PR[91] R[100]mm/sec CNT100;
   1:  PR[GP1:91,1] = PR[GP1:90,1] + -19.216;
   1:  PR[GP1:91,2] = PR[GP1:90,2] + -36.365;
   1:L PR[91] R[100]mm/sec CNT100;
   1:  PR[GP1:91,1] = PR[GP1:90,1] + -16.283;
   1:  PR[GP1:91,2] = PR[GP1:90,2] + -35.431;
   1:L PR[91] R[100]mm/sec CNT100;
   1:  PR[GP1:91,1] = PR[GP1:90,1] + -8.901;
   1:  PR[GP1:91,2] = PR[GP1:90,2] + -32.866;
   1:L PR[91] R[100]mm/sec CNT100;
   1:  PR[GP1:91,1] = PR[GP1:90,1] + -6.491;
   1:  PR[GP1:91,2] = PR[GP1:90,2] + -31.605;
   1:L PR[91] R[100]mm/sec CNT100;
   1:  PR[GP1:91,1] = PR[GP1:90,1] + -2.910;
   1:  PR[GP1:91,2] = PR[GP1:90,2] + -29.003;
   1:L PR[91] R[100]mm/sec CNT100;
   1:  PR[GP1:91,1] = PR[GP1:90,1] + -2.236;
   1:  PR[GP1:91,2] = PR[GP1:90,2] + -28.976;
   1:L PR[91] R[100]mm/sec CNT100;
   1:  PR[GP1:91,1] = PR[GP1:90,1] + 1.542;
   1:  PR[GP1:91,2] = PR[GP1:90,2] + -28.170;
   1:L PR[91] R[100]mm/sec CNT100;
   1:  PR[GP1:91,1] = PR[GP1:90,1] + 1.784;
   1:  PR[GP1:91,2] = PR[GP1:90,2] + -28.365;
   1:L PR[91] R[100]mm/sec CNT100;
   1:  PR[GP1:91,1] = PR[GP1:90,1] + 3.225;
   1:  PR[GP1:91,2] = PR[GP1:90,2] + -29.082;
   1:L PR[91] R[100]mm/sec CNT100;
   1:  PR[GP1:91,1] = PR[GP1:90,1] + 6.708;
   1:  PR[GP1:91,2] = PR[GP1:90,2] + -31.612;
   1:L PR[91] R[100]mm/sec CNT100;
   1:  PR[GP1:91,1] = PR[GP1:90,1] + 9.096;
   1:  PR[GP1:91,2] = PR[GP1:90,2] + -32.859;
   1:L PR[91] R[100]mm/sec CNT100;
   1:  PR[GP1:91,1] = PR[GP1:90,1] + 12.078;
   1:  PR[GP1:91,2] = PR[GP1:90,2] + -33.817;
   1:L PR[91] R[100]mm/sec CNT100;
   1:  PR[GP1:91,1] = PR[GP1:90,1] + 19.432;
   1:  PR[GP1:91,2] = PR[GP1:90,2] + -36.363;
   1:L PR[91] R[100]mm/sec CNT100;
   1:  PR[GP1:91,1] = PR[GP1:90,1] + 22.831;
   1:  PR[GP1:91,2] = PR[GP1:90,2] + -36.810;
   1:L PR[91] R[100]mm/sec CNT100;
   1:  PR[GP1:91,1] = PR[GP1:90,1] + 26.821;
   1:  PR[GP1:91,2] = PR[GP1:90,2] + -36.676;
   1:L PR[91] R[100]mm/sec CNT100;
   1:  PR[GP1:91,1] = PR[GP1:90,1] + 33.173;
   1:  PR[GP1:91,2] = PR[GP1:90,2] + -36.648;
   1:L PR[91] R[100]mm/sec CNT100;
   1:  PR[GP1:91,1] = PR[GP1:90,1] + 37.293;
   1:  PR[GP1:91,2] = PR[GP1:90,2] + -35.761;
   1:L PR[91] R[100]mm/sec CNT100;
   1:  PR[GP1:91,1] = PR[GP1:90,1] + 41.830;
   1:  PR[GP1:91,2] = PR[GP1:90,2] + -33.974;
   1:L PR[91] R[100]mm/sec CNT100;
   1:  PR[GP1:91,1] = PR[GP1:90,1] + 46.227;
   1:  PR[GP1:91,2] = PR[GP1:90,2] + -32.415;
   1:L PR[91] R[100]mm/sec CNT100;
   1:  PR[GP1:91,1] = PR[GP1:90,1] + 50.418;
   1:  PR[GP1:91,2] = PR[GP1:90,2] + -29.817;
   1:L PR[91] R[100]mm/sec CNT100;
   1:  PR[GP1:91,1] = PR[GP1:90,1] + 54.499;
   1:  PR[GP1:91,2] = PR[GP1:90,2] + -26.204;
   1:L PR[91] R[100]mm/sec CNT100;
   1:  PR[GP1:91,1] = PR[GP1:90,1] + 56.917;
   1:  PR[GP1:91,2] = PR[GP1:90,2] + -24.247;
   1:L PR[91] R[100]mm/sec CNT100;
   1:  PR[GP1:91,1] = PR[GP1:90,1] + 60.263;
   1:  PR[GP1:91,2] = PR[GP1:90,2] + -19.902;
   1:L PR[91] R[100]mm/sec CNT100;
   1:  PR[GP1:91,1] = PR[GP1:90,1] + 63.054;
   1:  PR[GP1:91,2] = PR[GP1:90,2] + -14.546;
   1:L PR[91] R[100]mm/sec CNT100;
   1:  PR[GP1:91,1] = PR[GP1:90,1] + 64.088;
   1:  PR[GP1:91,2] = PR[GP1:90,2] + -12.824;
   1:L PR[91] R[100]mm/sec CNT100;
   1:  PR[GP1:91,1] = PR[GP1:90,1] + 65.677;
   1:  PR[GP1:91,2] = PR[GP1:90,2] + -7.507;
   1:L PR[91] R[100]mm/sec CNT100;
   1:  PR[GP1:91,1] = PR[GP1:90,1] + 66.228;
   1:  PR[GP1:91,2] = PR[GP1:90,2] + -1.613;
   1:L PR[91] R[100]mm/sec CNT100;
   1:  PR[GP1:91,1] = PR[GP1:90,1] + 66.516;
   1:  PR[GP1:91,2] = PR[GP1:90,2] + -0.045;
   1:L PR[91] R[100]mm/sec CNT100;
   1:  PR[GP1:91,1] = PR[GP1:90,1] + 65.984;
   1:  PR[GP1:91,2] = PR[GP1:90,2] + 5.720;
   1:L PR[91] R[100]mm/sec CNT100;
   1:  PR[GP1:91,1] = PR[GP1:90,1] + 65.685;
   1:  PR[GP1:91,2] = PR[GP1:90,2] + 7.336;
   1:L PR[91] R[100]mm/sec CNT100;
   1:  PR[GP1:91,1] = PR[GP1:90,1] + 64.083;
   1:  PR[GP1:91,2] = PR[GP1:90,2] + 12.698;
   1:L PR[91] R[100]mm/sec CNT100;
   1:  PR[GP1:91,1] = PR[GP1:90,1] + 61.480;
   1:  PR[GP1:91,2] = PR[GP1:90,2] + 17.742;
   1:L PR[91] R[100]mm/sec CNT100;
   1:  PR[GP1:91,1] = PR[GP1:90,1] + 60.276;
   1:  PR[GP1:91,2] = PR[GP1:90,2] + 19.742;
   1:L PR[91] R[100]mm/sec CNT100;
   1:  PR[GP1:91,1] = PR[GP1:90,1] + 56.909;
   1:  PR[GP1:91,2] = PR[GP1:90,2] + 24.113;
   1:L PR[91] R[100]mm/sec CNT100;
   1:  PR[GP1:91,1] = PR[GP1:90,1] + 53.186;
   1:  PR[GP1:91,2] = PR[GP1:90,2] + 27.442;
   1:L PR[91] R[100]mm/sec CNT100;
   1:  PR[GP1:91,1] = PR[GP1:90,1] + 50.433;
   1:  PR[GP1:91,2] = PR[GP1:90,2] + 29.664;
   1:L PR[91] R[100]mm/sec CNT100;
   1:  PR[GP1:91,1] = PR[GP1:90,1] + 46.220;
   1:  PR[GP1:91,2] = PR[GP1:90,2] + 32.276;
   1:L PR[91] R[100]mm/sec CNT100;
   1:  PR[GP1:91,1] = PR[GP1:90,1] + 42.070;
   1:  PR[GP1:91,2] = PR[GP1:90,2] + 33.933;
   1:L PR[91] R[100]mm/sec CNT100;
   1:  PR[GP1:91,1] = PR[GP1:90,1] + 37.310;
   1:  PR[GP1:91,2] = PR[GP1:90,2] + 35.614;
   1:L PR[91] R[100]mm/sec CNT100;
   1:  PR[GP1:91,1] = PR[GP1:90,1] + 33.170;
   1:  PR[GP1:91,2] = PR[GP1:90,2] + 36.505;
   1:L PR[91] R[100]mm/sec CNT100;
   1:  PR[GP1:91,1] = PR[GP1:90,1] + 29.430;
   1:  PR[GP1:91,2] = PR[GP1:90,2] + 36.646;
   1:L PR[91] R[100]mm/sec CNT100;
   1:  PR[GP1:91,1] = PR[GP1:90,1] + 22.851;
   1:  PR[GP1:91,2] = PR[GP1:90,2] + 36.669;
   1:L PR[91] R[100]mm/sec CNT100;
   1:  PR[GP1:91,1] = PR[GP1:90,1] + 19.436;
   1:  PR[GP1:91,2] = PR[GP1:90,2] + 36.220;
   1:L PR[91] R[100]mm/sec CNT100;
   1:  PR[GP1:91,1] = PR[GP1:90,1] + 16.499;
   1:  PR[GP1:91,2] = PR[GP1:90,2] + 35.286;
   1:L PR[91] R[100]mm/sec CNT100;
   1:  PR[GP1:91,1] = PR[GP1:90,1] + 9.115;
   1:  PR[GP1:91,2] = PR[GP1:90,2] + 32.725;
   1:L PR[91] R[100]mm/sec CNT100;
   1:  PR[GP1:91,1] = PR[GP1:90,1] + 6.712;
   1:  PR[GP1:91,2] = PR[GP1:90,2] + 31.471;
   1:L PR[91] R[100]mm/sec CNT100;
   1:  PR[GP1:91,1] = PR[GP1:90,1] + 3.229;
   1:  PR[GP1:91,2] = PR[GP1:90,2] + 29.010;
   1:L PR[91] R[100]mm/sec CNT100;
   1:  PR[GP1:91,1] = PR[GP1:90,1] + 1.520;
   1:  PR[GP1:91,2] = PR[GP1:90,2] + 28.059;
   1:L PR[91] R[100]mm/sec CNT100;
   1:  ! -- Layer/Ebene 95 -- !;
   1:  PR[91] = PR[90];
   1:  PR[GP1:91,1] = PR[GP1:90,1] + 0.453;
   1:  PR[GP1:91,2] = PR[GP1:90,2] + 28.392;
   1:  PR[GP1:91,3] = PR[GP1:90,3] + 58.255;
   1:L PR[91] R[100]mm/sec CNT100;
   1:  PR[GP1:91,1] = PR[GP1:90,1] + -2.924;
   1:  PR[GP1:91,2] = PR[GP1:90,2] + 29.177;
   1:L PR[91] R[100]mm/sec CNT100;
   1:  PR[GP1:91,1] = PR[GP1:90,1] + -6.284;
   1:  PR[GP1:91,2] = PR[GP1:90,2] + 31.551;
   1:L PR[91] R[100]mm/sec CNT100;
   1:  PR[GP1:91,1] = PR[GP1:90,1] + -8.566;
   1:  PR[GP1:91,2] = PR[GP1:90,2] + 32.745;
   1:L PR[91] R[100]mm/sec CNT100;
   1:  PR[GP1:91,1] = PR[GP1:90,1] + -11.389;
   1:  PR[GP1:91,2] = PR[GP1:90,2] + 33.652;
   1:L PR[91] R[100]mm/sec CNT100;
   1:  PR[GP1:91,1] = PR[GP1:90,1] + -19.036;
   1:  PR[GP1:91,2] = PR[GP1:90,2] + 36.296;
   1:L PR[91] R[100]mm/sec CNT100;
   1:  PR[GP1:91,1] = PR[GP1:90,1] + -22.287;
   1:  PR[GP1:91,2] = PR[GP1:90,2] + 36.720;
   1:L PR[91] R[100]mm/sec CNT100;
   1:  PR[GP1:91,1] = PR[GP1:90,1] + -26.120;
   1:  PR[GP1:91,2] = PR[GP1:90,2] + 36.589;
   1:L PR[91] R[100]mm/sec CNT100;
   1:  PR[GP1:91,1] = PR[GP1:90,1] + -32.806;
   1:  PR[GP1:91,2] = PR[GP1:90,2] + 36.555;
   1:L PR[91] R[100]mm/sec CNT100;
   1:  PR[GP1:91,1] = PR[GP1:90,1] + -36.774;
   1:  PR[GP1:91,2] = PR[GP1:90,2] + 35.699;
   1:L PR[91] R[100]mm/sec CNT100;
   1:  PR[GP1:91,1] = PR[GP1:90,1] + -41.135;
   1:  PR[GP1:91,2] = PR[GP1:90,2] + 33.972;
   1:L PR[91] R[100]mm/sec CNT100;
   1:  PR[GP1:91,1] = PR[GP1:90,1] + -45.858;
   1:  PR[GP1:91,2] = PR[GP1:90,2] + 32.295;
   1:L PR[91] R[100]mm/sec CNT100;
   1:  PR[GP1:91,1] = PR[GP1:90,1] + -49.934;
   1:  PR[GP1:91,2] = PR[GP1:90,2] + 29.756;
   1:L PR[91] R[100]mm/sec CNT100;
   1:  PR[GP1:91,1] = PR[GP1:90,1] + -53.902;
   1:  PR[GP1:91,2] = PR[GP1:90,2] + 26.233;
   1:L PR[91] R[100]mm/sec CNT100;
   1:  PR[GP1:91,1] = PR[GP1:90,1] + -56.589;
   1:  PR[GP1:91,2] = PR[GP1:90,2] + 24.059;
   1:L PR[91] R[100]mm/sec CNT100;
   1:  PR[GP1:91,1] = PR[GP1:90,1] + -59.800;
   1:  PR[GP1:91,2] = PR[GP1:90,2] + 19.879;
   1:L PR[91] R[100]mm/sec CNT100;
   1:  PR[GP1:91,1] = PR[GP1:90,1] + -62.499;
   1:  PR[GP1:91,2] = PR[GP1:90,2] + 14.641;
   1:L PR[91] R[100]mm/sec CNT100;
   1:  PR[GP1:91,1] = PR[GP1:90,1] + -63.712;
   1:  PR[GP1:91,2] = PR[GP1:90,2] + 12.616;
   1:L PR[91] R[100]mm/sec CNT100;
   1:  PR[GP1:91,1] = PR[GP1:90,1] + -65.257;
   1:  PR[GP1:91,2] = PR[GP1:90,2] + 7.374;
   1:L PR[91] R[100]mm/sec CNT100;
   1:  PR[GP1:91,1] = PR[GP1:90,1] + -65.767;
   1:  PR[GP1:91,2] = PR[GP1:90,2] + 1.801;
   1:L PR[91] R[100]mm/sec CNT100;
   1:  PR[GP1:91,1] = PR[GP1:90,1] + -66.117;
   1:  PR[GP1:91,2] = PR[GP1:90,2] + -0.100;
   1:L PR[91] R[100]mm/sec CNT100;
   1:  PR[GP1:91,1] = PR[GP1:90,1] + -65.624;
   1:  PR[GP1:91,2] = PR[GP1:90,2] + -5.552;
   1:L PR[91] R[100]mm/sec CNT100;
   1:  PR[GP1:91,1] = PR[GP1:90,1] + -65.264;
   1:  PR[GP1:91,2] = PR[GP1:90,2] + -7.492;
   1:L PR[91] R[100]mm/sec CNT100;
   1:  PR[GP1:91,1] = PR[GP1:90,1] + -63.706;
   1:  PR[GP1:91,2] = PR[GP1:90,2] + -12.780;
   1:L PR[91] R[100]mm/sec CNT100;
   1:  PR[GP1:91,1] = PR[GP1:90,1] + -61.185;
   1:  PR[GP1:91,2] = PR[GP1:90,2] + -17.723;
   1:L PR[91] R[100]mm/sec CNT100;
   1:  PR[GP1:91,1] = PR[GP1:90,1] + -59.810;
   1:  PR[GP1:91,2] = PR[GP1:90,2] + -20.009;
   1:L PR[91] R[100]mm/sec CNT100;
   1:  PR[GP1:91,1] = PR[GP1:90,1] + -56.578;
   1:  PR[GP1:91,2] = PR[GP1:90,2] + -24.216;
   1:L PR[91] R[100]mm/sec CNT100;
   1:  PR[GP1:91,1] = PR[GP1:90,1] + -52.948;
   1:  PR[GP1:91,2] = PR[GP1:90,2] + -27.472;
   1:L PR[91] R[100]mm/sec CNT100;
   1:  PR[GP1:91,1] = PR[GP1:90,1] + -49.943;
   1:  PR[GP1:91,2] = PR[GP1:90,2] + -29.895;
   1:L PR[91] R[100]mm/sec CNT100;
   1:  PR[GP1:91,1] = PR[GP1:90,1] + -45.844;
   1:  PR[GP1:91,2] = PR[GP1:90,2] + -32.448;
   1:L PR[91] R[100]mm/sec CNT100;
   1:  PR[GP1:91,1] = PR[GP1:90,1] + -41.837;
   1:  PR[GP1:91,2] = PR[GP1:90,2] + -34.057;
   1:L PR[91] R[100]mm/sec CNT100;
   1:  PR[GP1:91,1] = PR[GP1:90,1] + -36.778;
   1:  PR[GP1:91,2] = PR[GP1:90,2] + -35.842;
   1:L PR[91] R[100]mm/sec CNT100;
   1:  PR[GP1:91,1] = PR[GP1:90,1] + -32.788;
   1:  PR[GP1:91,2] = PR[GP1:90,2] + -36.703;
   1:L PR[91] R[100]mm/sec CNT100;
   1:  PR[GP1:91,1] = PR[GP1:90,1] + -29.172;
   1:  PR[GP1:91,2] = PR[GP1:90,2] + -36.842;
   1:L PR[91] R[100]mm/sec CNT100;
   1:  PR[GP1:91,1] = PR[GP1:90,1] + -22.285;
   1:  PR[GP1:91,2] = PR[GP1:90,2] + -36.864;
   1:L PR[91] R[100]mm/sec CNT100;
   1:  PR[GP1:91,1] = PR[GP1:90,1] + -19.017;
   1:  PR[GP1:91,2] = PR[GP1:90,2] + -36.437;
   1:L PR[91] R[100]mm/sec CNT100;
   1:  PR[GP1:91,1] = PR[GP1:90,1] + -16.215;
   1:  PR[GP1:91,2] = PR[GP1:90,2] + -35.545;
   1:L PR[91] R[100]mm/sec CNT100;
   1:  PR[GP1:91,1] = PR[GP1:90,1] + -8.559;
   1:  PR[GP1:91,2] = PR[GP1:90,2] + -32.885;
   1:L PR[91] R[100]mm/sec CNT100;
   1:  PR[GP1:91,1] = PR[GP1:90,1] + -6.280;
   1:  PR[GP1:91,2] = PR[GP1:90,2] + -31.692;
   1:L PR[91] R[100]mm/sec CNT100;
   1:  PR[GP1:91,1] = PR[GP1:90,1] + -2.882;
   1:  PR[GP1:91,2] = PR[GP1:90,2] + -29.223;
   1:L PR[91] R[100]mm/sec CNT100;
   1:  PR[GP1:91,1] = PR[GP1:90,1] + -2.070;
   1:  PR[GP1:91,2] = PR[GP1:90,2] + -29.191;
   1:L PR[91] R[100]mm/sec CNT100;
   1:  PR[GP1:91,1] = PR[GP1:90,1] + 1.572;
   1:  PR[GP1:91,2] = PR[GP1:90,2] + -28.414;
   1:L PR[91] R[100]mm/sec CNT100;
   1:  PR[GP1:91,1] = PR[GP1:90,1] + 1.832;
   1:  PR[GP1:91,2] = PR[GP1:90,2] + -28.623;
   1:L PR[91] R[100]mm/sec CNT100;
   1:  PR[GP1:91,1] = PR[GP1:90,1] + 3.197;
   1:  PR[GP1:91,2] = PR[GP1:90,2] + -29.302;
   1:L PR[91] R[100]mm/sec CNT100;
   1:  PR[GP1:91,1] = PR[GP1:90,1] + 6.496;
   1:  PR[GP1:91,2] = PR[GP1:90,2] + -31.699;
   1:L PR[91] R[100]mm/sec CNT100;
   1:  PR[GP1:91,1] = PR[GP1:90,1] + 8.754;
   1:  PR[GP1:91,2] = PR[GP1:90,2] + -32.878;
   1:L PR[91] R[100]mm/sec CNT100;
   1:  PR[GP1:91,1] = PR[GP1:90,1] + 11.576;
   1:  PR[GP1:91,2] = PR[GP1:90,2] + -33.784;
   1:L PR[91] R[100]mm/sec CNT100;
   1:  PR[GP1:91,1] = PR[GP1:90,1] + 19.233;
   1:  PR[GP1:91,2] = PR[GP1:90,2] + -36.435;
   1:L PR[91] R[100]mm/sec CNT100;
   1:  PR[GP1:91,1] = PR[GP1:90,1] + 22.480;
   1:  PR[GP1:91,2] = PR[GP1:90,2] + -36.862;
   1:L PR[91] R[100]mm/sec CNT100;
   1:  PR[GP1:91,1] = PR[GP1:90,1] + 26.294;
   1:  PR[GP1:91,2] = PR[GP1:90,2] + -36.734;
   1:L PR[91] R[100]mm/sec CNT100;
   1:  PR[GP1:91,1] = PR[GP1:90,1] + 32.986;
   1:  PR[GP1:91,2] = PR[GP1:90,2] + -36.704;
   1:L PR[91] R[100]mm/sec CNT100;
   1:  PR[GP1:91,1] = PR[GP1:90,1] + 36.948;
   1:  PR[GP1:91,2] = PR[GP1:90,2] + -35.852;
   1:L PR[91] R[100]mm/sec CNT100;
   1:  PR[GP1:91,1] = PR[GP1:90,1] + 41.315;
   1:  PR[GP1:91,2] = PR[GP1:90,2] + -34.131;
   1:L PR[91] R[100]mm/sec CNT100;
   1:  PR[GP1:91,1] = PR[GP1:90,1] + 46.044;
   1:  PR[GP1:91,2] = PR[GP1:90,2] + -32.455;
   1:L PR[91] R[100]mm/sec CNT100;
   1:  PR[GP1:91,1] = PR[GP1:90,1] + 50.095;
   1:  PR[GP1:91,2] = PR[GP1:90,2] + -29.944;
   1:L PR[91] R[100]mm/sec CNT100;
   1:  PR[GP1:91,1] = PR[GP1:90,1] + 54.041;
   1:  PR[GP1:91,2] = PR[GP1:90,2] + -26.450;
   1:L PR[91] R[100]mm/sec CNT100;
   1:  PR[GP1:91,1] = PR[GP1:90,1] + 56.735;
   1:  PR[GP1:91,2] = PR[GP1:90,2] + -24.269;
   1:L PR[91] R[100]mm/sec CNT100;
   1:  PR[GP1:91,1] = PR[GP1:90,1] + 59.980;
   1:  PR[GP1:91,2] = PR[GP1:90,2] + -20.057;
   1:L PR[91] R[100]mm/sec CNT100;
   1:  PR[GP1:91,1] = PR[GP1:90,1] + 62.687;
   1:  PR[GP1:91,2] = PR[GP1:90,2] + -14.862;
   1:L PR[91] R[100]mm/sec CNT100;
   1:  PR[GP1:91,1] = PR[GP1:90,1] + 63.902;
   1:  PR[GP1:91,2] = PR[GP1:90,2] + -12.838;
   1:L PR[91] R[100]mm/sec CNT100;
   1:  PR[GP1:91,1] = PR[GP1:90,1] + 65.445;
   1:  PR[GP1:91,2] = PR[GP1:90,2] + -7.674;
   1:L PR[91] R[100]mm/sec CNT100;
   1:  PR[GP1:91,1] = PR[GP1:90,1] + 65.980;
   1:  PR[GP1:91,2] = PR[GP1:90,2] + -1.948;
   1:L PR[91] R[100]mm/sec CNT100;
   1:  PR[GP1:91,1] = PR[GP1:90,1] + 66.330;
   1:  PR[GP1:91,2] = PR[GP1:90,2] + -0.045;
   1:L PR[91] R[100]mm/sec CNT100;
   1:  PR[GP1:91,1] = PR[GP1:90,1] + 65.813;
   1:  PR[GP1:91,2] = PR[GP1:90,2] + 5.559;
   1:L PR[91] R[100]mm/sec CNT100;
   1:  PR[GP1:91,1] = PR[GP1:90,1] + 65.453;
   1:  PR[GP1:91,2] = PR[GP1:90,2] + 7.504;
   1:L PR[91] R[100]mm/sec CNT100;
   1:  PR[GP1:91,1] = PR[GP1:90,1] + 63.896;
   1:  PR[GP1:91,2] = PR[GP1:90,2] + 12.712;
   1:L PR[91] R[100]mm/sec CNT100;
   1:  PR[GP1:91,1] = PR[GP1:90,1] + 61.368;
   1:  PR[GP1:91,2] = PR[GP1:90,2] + 17.612;
   1:L PR[91] R[100]mm/sec CNT100;
   1:  PR[GP1:91,1] = PR[GP1:90,1] + 59.992;
   1:  PR[GP1:91,2] = PR[GP1:90,2] + 19.897;
   1:L PR[91] R[100]mm/sec CNT100;
   1:  PR[GP1:91,1] = PR[GP1:90,1] + 56.728;
   1:  PR[GP1:91,2] = PR[GP1:90,2] + 24.135;
   1:L PR[91] R[100]mm/sec CNT100;
   1:  PR[GP1:91,1] = PR[GP1:90,1] + 53.117;
   1:  PR[GP1:91,2] = PR[GP1:90,2] + 27.364;
   1:L PR[91] R[100]mm/sec CNT100;
   1:  PR[GP1:91,1] = PR[GP1:90,1] + 50.110;
   1:  PR[GP1:91,2] = PR[GP1:90,2] + 29.791;
   1:L PR[91] R[100]mm/sec CNT100;
   1:  PR[GP1:91,1] = PR[GP1:90,1] + 46.038;
   1:  PR[GP1:91,2] = PR[GP1:90,2] + 32.315;
   1:L PR[91] R[100]mm/sec CNT100;
   1:  PR[GP1:91,1] = PR[GP1:90,1] + 42.026;
   1:  PR[GP1:91,2] = PR[GP1:90,2] + 33.918;
   1:L PR[91] R[100]mm/sec CNT100;
   1:  PR[GP1:91,1] = PR[GP1:90,1] + 36.965;
   1:  PR[GP1:91,2] = PR[GP1:90,2] + 35.704;
   1:L PR[91] R[100]mm/sec CNT100;
   1:  PR[GP1:91,1] = PR[GP1:90,1] + 32.983;
   1:  PR[GP1:91,2] = PR[GP1:90,2] + 36.561;
   1:L PR[91] R[100]mm/sec CNT100;
   1:  PR[GP1:91,1] = PR[GP1:90,1] + 29.385;
   1:  PR[GP1:91,2] = PR[GP1:90,2] + 36.697;
   1:L PR[91] R[100]mm/sec CNT100;
   1:  PR[GP1:91,1] = PR[GP1:90,1] + 22.500;
   1:  PR[GP1:91,2] = PR[GP1:90,2] + 36.721;
   1:L PR[91] R[100]mm/sec CNT100;
   1:  PR[GP1:91,1] = PR[GP1:90,1] + 19.238;
   1:  PR[GP1:91,2] = PR[GP1:90,2] + 36.292;
   1:L PR[91] R[100]mm/sec CNT100;
   1:  PR[GP1:91,1] = PR[GP1:90,1] + 16.431;
   1:  PR[GP1:91,2] = PR[GP1:90,2] + 35.399;
   1:L PR[91] R[100]mm/sec CNT100;
   1:  PR[GP1:91,1] = PR[GP1:90,1] + 8.773;
   1:  PR[GP1:91,2] = PR[GP1:90,2] + 32.744;
   1:L PR[91] R[100]mm/sec CNT100;
   1:  PR[GP1:91,1] = PR[GP1:90,1] + 6.500;
   1:  PR[GP1:91,2] = PR[GP1:90,2] + 31.558;
   1:L PR[91] R[100]mm/sec CNT100;
   1:  PR[GP1:91,1] = PR[GP1:90,1] + 3.202;
   1:  PR[GP1:91,2] = PR[GP1:90,2] + 29.222;
   1:L PR[91] R[100]mm/sec CNT100;
   1:  PR[GP1:91,1] = PR[GP1:90,1] + 1.550;
   1:  PR[GP1:91,2] = PR[GP1:90,2] + 28.302;
   1:L PR[91] R[100]mm/sec CNT100;
   1:  ! -- Layer/Ebene 96 -- !;
   1:  PR[91] = PR[90];
   1:  PR[GP1:91,1] = PR[GP1:90,1] + 0.302;
   1:  PR[GP1:91,2] = PR[GP1:90,2] + 28.650;
   1:  PR[GP1:91,3] = PR[GP1:90,3] + 58.865;
   1:L PR[91] R[100]mm/sec CNT100;
   1:  PR[GP1:91,1] = PR[GP1:90,1] + -2.897;
   1:  PR[GP1:91,2] = PR[GP1:90,2] + 29.394;
   1:L PR[91] R[100]mm/sec CNT100;
   1:  PR[GP1:91,1] = PR[GP1:90,1] + -6.074;
   1:  PR[GP1:91,2] = PR[GP1:90,2] + 31.639;
   1:L PR[91] R[100]mm/sec CNT100;
   1:  PR[GP1:91,1] = PR[GP1:90,1] + -8.224;
   1:  PR[GP1:91,2] = PR[GP1:90,2] + 32.764;
   1:L PR[91] R[100]mm/sec CNT100;
   1:  PR[GP1:91,1] = PR[GP1:90,1] + -10.889;
   1:  PR[GP1:91,2] = PR[GP1:90,2] + 33.620;
   1:L PR[91] R[100]mm/sec CNT100;
   1:  PR[GP1:91,1] = PR[GP1:90,1] + -18.838;
   1:  PR[GP1:91,2] = PR[GP1:90,2] + 36.368;
   1:L PR[91] R[100]mm/sec CNT100;
   1:  PR[GP1:91,1] = PR[GP1:90,1] + -21.936;
   1:  PR[GP1:91,2] = PR[GP1:90,2] + 36.773;
   1:L PR[91] R[100]mm/sec CNT100;
   1:  PR[GP1:91,1] = PR[GP1:90,1] + -25.591;
   1:  PR[GP1:91,2] = PR[GP1:90,2] + 36.647;
   1:L PR[91] R[100]mm/sec CNT100;
   1:  PR[GP1:91,1] = PR[GP1:90,1] + -32.618;
   1:  PR[GP1:91,2] = PR[GP1:90,2] + 36.612;
   1:L PR[91] R[100]mm/sec CNT100;
   1:  PR[GP1:91,1] = PR[GP1:90,1] + -36.428;
   1:  PR[GP1:91,2] = PR[GP1:90,2] + 35.790;
   1:L PR[91] R[100]mm/sec CNT100;
   1:  PR[GP1:91,1] = PR[GP1:90,1] + -40.619;
   1:  PR[GP1:91,2] = PR[GP1:90,2] + 34.131;
   1:L PR[91] R[100]mm/sec CNT100;
   1:  PR[GP1:91,1] = PR[GP1:90,1] + -45.675;
   1:  PR[GP1:91,2] = PR[GP1:90,2] + 32.335;
   1:L PR[91] R[100]mm/sec CNT100;
   1:  PR[GP1:91,1] = PR[GP1:90,1] + -49.609;
   1:  PR[GP1:91,2] = PR[GP1:90,2] + 29.884;
   1:L PR[91] R[100]mm/sec CNT100;
   1:  PR[GP1:91,1] = PR[GP1:90,1] + -53.442;
   1:  PR[GP1:91,2] = PR[GP1:90,2] + 26.481;
   1:L PR[91] R[100]mm/sec CNT100;
   1:  PR[GP1:91,1] = PR[GP1:90,1] + -56.405;
   1:  PR[GP1:91,2] = PR[GP1:90,2] + 24.083;
   1:L PR[91] R[100]mm/sec CNT100;
   1:  PR[GP1:91,1] = PR[GP1:90,1] + -59.515;
   1:  PR[GP1:91,2] = PR[GP1:90,2] + 20.035;
   1:L PR[91] R[100]mm/sec CNT100;
   1:  PR[GP1:91,1] = PR[GP1:90,1] + -62.131;
   1:  PR[GP1:91,2] = PR[GP1:90,2] + 14.960;
   1:L PR[91] R[100]mm/sec CNT100;
   1:  PR[GP1:91,1] = PR[GP1:90,1] + -63.525;
   1:  PR[GP1:91,2] = PR[GP1:90,2] + 12.631;
   1:L PR[91] R[100]mm/sec CNT100;
   1:  PR[GP1:91,1] = PR[GP1:90,1] + -65.024;
   1:  PR[GP1:91,2] = PR[GP1:90,2] + 7.546;
   1:L PR[91] R[100]mm/sec CNT100;
   1:  PR[GP1:91,1] = PR[GP1:90,1] + -65.519;
   1:  PR[GP1:91,2] = PR[GP1:90,2] + 2.136;
   1:L PR[91] R[100]mm/sec CNT100;
   1:  PR[GP1:91,1] = PR[GP1:90,1] + -65.931;
   1:  PR[GP1:91,2] = PR[GP1:90,2] + -0.100;
   1:L PR[91] R[100]mm/sec CNT100;
   1:  PR[GP1:91,1] = PR[GP1:90,1] + -65.452;
   1:  PR[GP1:91,2] = PR[GP1:90,2] + -5.396;
   1:L PR[91] R[100]mm/sec CNT100;
   1:  PR[GP1:91,1] = PR[GP1:90,1] + -65.031;
   1:  PR[GP1:91,2] = PR[GP1:90,2] + -7.664;
   1:L PR[91] R[100]mm/sec CNT100;
   1:  PR[GP1:91,1] = PR[GP1:90,1] + -63.518;
   1:  PR[GP1:91,2] = PR[GP1:90,2] + -12.796;
   1:L PR[91] R[100]mm/sec CNT100;
   1:  PR[GP1:91,1] = PR[GP1:90,1] + -61.072;
   1:  PR[GP1:91,2] = PR[GP1:90,2] + -17.593;
   1:L PR[91] R[100]mm/sec CNT100;
   1:  PR[GP1:91,1] = PR[GP1:90,1] + -59.526;
   1:  PR[GP1:91,2] = PR[GP1:90,2] + -20.165;
   1:L PR[91] R[100]mm/sec CNT100;
   1:  PR[GP1:91,1] = PR[GP1:90,1] + -56.395;
   1:  PR[GP1:91,2] = PR[GP1:90,2] + -24.241;
   1:L PR[91] R[100]mm/sec CNT100;
   1:  PR[GP1:91,1] = PR[GP1:90,1] + -52.878;
   1:  PR[GP1:91,2] = PR[GP1:90,2] + -27.395;
   1:L PR[91] R[100]mm/sec CNT100;
   1:  PR[GP1:91,1] = PR[GP1:90,1] + -49.618;
   1:  PR[GP1:91,2] = PR[GP1:90,2] + -30.023;
   1:L PR[91] R[100]mm/sec CNT100;
   1:  PR[GP1:91,1] = PR[GP1:90,1] + -45.660;
   1:  PR[GP1:91,2] = PR[GP1:90,2] + -32.488;
   1:L PR[91] R[100]mm/sec CNT100;
   1:  PR[GP1:91,1] = PR[GP1:90,1] + -41.791;
   1:  PR[GP1:91,2] = PR[GP1:90,2] + -34.042;
   1:L PR[91] R[100]mm/sec CNT100;
   1:  PR[GP1:91,1] = PR[GP1:90,1] + -36.431;
   1:  PR[GP1:91,2] = PR[GP1:90,2] + -35.933;
   1:L PR[91] R[100]mm/sec CNT100;
   1:  PR[GP1:91,1] = PR[GP1:90,1] + -32.600;
   1:  PR[GP1:91,2] = PR[GP1:90,2] + -36.759;
   1:L PR[91] R[100]mm/sec CNT100;
   1:  PR[GP1:91,1] = PR[GP1:90,1] + -29.127;
   1:  PR[GP1:91,2] = PR[GP1:90,2] + -36.893;
   1:L PR[91] R[100]mm/sec CNT100;
   1:  PR[GP1:91,1] = PR[GP1:90,1] + -21.933;
   1:  PR[GP1:91,2] = PR[GP1:90,2] + -36.916;
   1:L PR[91] R[100]mm/sec CNT100;
   1:  PR[GP1:91,1] = PR[GP1:90,1] + -18.818;
   1:  PR[GP1:91,2] = PR[GP1:90,2] + -36.509;
   1:L PR[91] R[100]mm/sec CNT100;
   1:  PR[GP1:91,1] = PR[GP1:90,1] + -16.146;
   1:  PR[GP1:91,2] = PR[GP1:90,2] + -35.659;
   1:L PR[91] R[100]mm/sec CNT100;
   1:  PR[GP1:91,1] = PR[GP1:90,1] + -8.217;
   1:  PR[GP1:91,2] = PR[GP1:90,2] + -32.903;
   1:L PR[91] R[100]mm/sec CNT100;
   1:  PR[GP1:91,1] = PR[GP1:90,1] + -6.069;
   1:  PR[GP1:91,2] = PR[GP1:90,2] + -31.779;
   1:L PR[91] R[100]mm/sec CNT100;
   1:  PR[GP1:91,1] = PR[GP1:90,1] + -2.854;
   1:  PR[GP1:91,2] = PR[GP1:90,2] + -29.443;
   1:L PR[91] R[100]mm/sec CNT100;
   1:  PR[GP1:91,1] = PR[GP1:90,1] + -1.905;
   1:  PR[GP1:91,2] = PR[GP1:90,2] + -29.406;
   1:L PR[91] R[100]mm/sec CNT100;
   1:  PR[GP1:91,1] = PR[GP1:90,1] + 1.603;
   1:  PR[GP1:91,2] = PR[GP1:90,2] + -28.657;
   1:L PR[91] R[100]mm/sec CNT100;
   1:  PR[GP1:91,1] = PR[GP1:90,1] + 1.881;
   1:  PR[GP1:91,2] = PR[GP1:90,2] + -28.881;
   1:L PR[91] R[100]mm/sec CNT100;
   1:  PR[GP1:91,1] = PR[GP1:90,1] + 3.169;
   1:  PR[GP1:91,2] = PR[GP1:90,2] + -29.522;
   1:L PR[91] R[100]mm/sec CNT100;
   1:  PR[GP1:91,1] = PR[GP1:90,1] + 6.285;
   1:  PR[GP1:91,2] = PR[GP1:90,2] + -31.786;
   1:L PR[91] R[100]mm/sec CNT100;
   1:  PR[GP1:91,1] = PR[GP1:90,1] + 8.412;
   1:  PR[GP1:91,2] = PR[GP1:90,2] + -32.896;
   1:L PR[91] R[100]mm/sec CNT100;
   1:  PR[GP1:91,1] = PR[GP1:90,1] + 11.075;
   1:  PR[GP1:91,2] = PR[GP1:90,2] + -33.752;
   1:L PR[91] R[100]mm/sec CNT100;
   1:  PR[GP1:91,1] = PR[GP1:90,1] + 19.035;
   1:  PR[GP1:91,2] = PR[GP1:90,2] + -36.508;
   1:L PR[91] R[100]mm/sec CNT100;
   1:  PR[GP1:91,1] = PR[GP1:90,1] + 22.128;
   1:  PR[GP1:91,2] = PR[GP1:90,2] + -36.914;
   1:L PR[91] R[100]mm/sec CNT100;
   1:  PR[GP1:91,1] = PR[GP1:90,1] + 25.766;
   1:  PR[GP1:91,2] = PR[GP1:90,2] + -36.792;
   1:L PR[91] R[100]mm/sec CNT100;
   1:  PR[GP1:91,1] = PR[GP1:90,1] + 32.799;
   1:  PR[GP1:91,2] = PR[GP1:90,2] + -36.761;
   1:L PR[91] R[100]mm/sec CNT100;
   1:  PR[GP1:91,1] = PR[GP1:90,1] + 36.603;
   1:  PR[GP1:91,2] = PR[GP1:90,2] + -35.942;
   1:L PR[91] R[100]mm/sec CNT100;
   1:  PR[GP1:91,1] = PR[GP1:90,1] + 40.799;
   1:  PR[GP1:91,2] = PR[GP1:90,2] + -34.289;
   1:L PR[91] R[100]mm/sec CNT100;
   1:  PR[GP1:91,1] = PR[GP1:90,1] + 45.861;
   1:  PR[GP1:91,2] = PR[GP1:90,2] + -32.495;
   1:L PR[91] R[100]mm/sec CNT100;
   1:  PR[GP1:91,1] = PR[GP1:90,1] + 49.771;
   1:  PR[GP1:91,2] = PR[GP1:90,2] + -30.071;
   1:L PR[91] R[100]mm/sec CNT100;
   1:  PR[GP1:91,1] = PR[GP1:90,1] + 53.582;
   1:  PR[GP1:91,2] = PR[GP1:90,2] + -26.696;
   1:L PR[91] R[100]mm/sec CNT100;
   1:  PR[GP1:91,1] = PR[GP1:90,1] + 56.554;
   1:  PR[GP1:91,2] = PR[GP1:90,2] + -24.291;
   1:L PR[91] R[100]mm/sec CNT100;
   1:  PR[GP1:91,1] = PR[GP1:90,1] + 59.696;
   1:  PR[GP1:91,2] = PR[GP1:90,2] + -20.212;
   1:L PR[91] R[100]mm/sec CNT100;
   1:  PR[GP1:91,1] = PR[GP1:90,1] + 62.319;
   1:  PR[GP1:91,2] = PR[GP1:90,2] + -15.178;
   1:L PR[91] R[100]mm/sec CNT100;
   1:  PR[GP1:91,1] = PR[GP1:90,1] + 63.715;
   1:  PR[GP1:91,2] = PR[GP1:90,2] + -12.852;
   1:L PR[91] R[100]mm/sec CNT100;
   1:  PR[GP1:91,1] = PR[GP1:90,1] + 65.212;
   1:  PR[GP1:91,2] = PR[GP1:90,2] + -7.842;
   1:L PR[91] R[100]mm/sec CNT100;
   1:  PR[GP1:91,1] = PR[GP1:90,1] + 65.732;
   1:  PR[GP1:91,2] = PR[GP1:90,2] + -2.283;
   1:L PR[91] R[100]mm/sec CNT100;
   1:  PR[GP1:91,1] = PR[GP1:90,1] + 66.144;
   1:  PR[GP1:91,2] = PR[GP1:90,2] + -0.045;
   1:L PR[91] R[100]mm/sec CNT100;
   1:  PR[GP1:91,1] = PR[GP1:90,1] + 65.641;
   1:  PR[GP1:91,2] = PR[GP1:90,2] + 5.399;
   1:L PR[91] R[100]mm/sec CNT100;
   1:  PR[GP1:91,1] = PR[GP1:90,1] + 65.220;
   1:  PR[GP1:91,2] = PR[GP1:90,2] + 7.671;
   1:L PR[91] R[100]mm/sec CNT100;
   1:  PR[GP1:91,1] = PR[GP1:90,1] + 63.710;
   1:  PR[GP1:91,2] = PR[GP1:90,2] + 12.726;
   1:L PR[91] R[100]mm/sec CNT100;
   1:  PR[GP1:91,1] = PR[GP1:90,1] + 61.256;
   1:  PR[GP1:91,2] = PR[GP1:90,2] + 17.481;
   1:L PR[91] R[100]mm/sec CNT100;
   1:  PR[GP1:91,1] = PR[GP1:90,1] + 59.708;
   1:  PR[GP1:91,2] = PR[GP1:90,2] + 20.052;
   1:L PR[91] R[100]mm/sec CNT100;
   1:  PR[GP1:91,1] = PR[GP1:90,1] + 56.546;
   1:  PR[GP1:91,2] = PR[GP1:90,2] + 24.157;
   1:L PR[91] R[100]mm/sec CNT100;
   1:  PR[GP1:91,1] = PR[GP1:90,1] + 53.048;
   1:  PR[GP1:91,2] = PR[GP1:90,2] + 27.285;
   1:L PR[91] R[100]mm/sec CNT100;
   1:  PR[GP1:91,1] = PR[GP1:90,1] + 49.786;
   1:  PR[GP1:91,2] = PR[GP1:90,2] + 29.918;
   1:L PR[91] R[100]mm/sec CNT100;
   1:  PR[GP1:91,1] = PR[GP1:90,1] + 45.855;
   1:  PR[GP1:91,2] = PR[GP1:90,2] + 32.355;
   1:L PR[91] R[100]mm/sec CNT100;
   1:  PR[GP1:91,1] = PR[GP1:90,1] + 41.981;
   1:  PR[GP1:91,2] = PR[GP1:90,2] + 33.902;
   1:L PR[91] R[100]mm/sec CNT100;
   1:  PR[GP1:91,1] = PR[GP1:90,1] + 36.621;
   1:  PR[GP1:91,2] = PR[GP1:90,2] + 35.795;
   1:L PR[91] R[100]mm/sec CNT100;
   1:  PR[GP1:91,1] = PR[GP1:90,1] + 32.797;
   1:  PR[GP1:91,2] = PR[GP1:90,2] + 36.618;
   1:L PR[91] R[100]mm/sec CNT100;
   1:  PR[GP1:91,1] = PR[GP1:90,1] + 29.340;
   1:  PR[GP1:91,2] = PR[GP1:90,2] + 36.748;
   1:L PR[91] R[100]mm/sec CNT100;
   1:  PR[GP1:91,1] = PR[GP1:90,1] + 22.149;
   1:  PR[GP1:91,2] = PR[GP1:90,2] + 36.773;
   1:L PR[91] R[100]mm/sec CNT100;
   1:  PR[GP1:91,1] = PR[GP1:90,1] + 19.039;
   1:  PR[GP1:91,2] = PR[GP1:90,2] + 36.365;
   1:L PR[91] R[100]mm/sec CNT100;
   1:  PR[GP1:91,1] = PR[GP1:90,1] + 16.364;
   1:  PR[GP1:91,2] = PR[GP1:90,2] + 35.513;
   1:L PR[91] R[100]mm/sec CNT100;
   1:  PR[GP1:91,1] = PR[GP1:90,1] + 8.432;
   1:  PR[GP1:91,2] = PR[GP1:90,2] + 32.763;
   1:L PR[91] R[100]mm/sec CNT100;
   1:  PR[GP1:91,1] = PR[GP1:90,1] + 6.289;
   1:  PR[GP1:91,2] = PR[GP1:90,2] + 31.645;
   1:L PR[91] R[100]mm/sec CNT100;
   1:  PR[GP1:91,1] = PR[GP1:90,1] + 3.174;
   1:  PR[GP1:91,2] = PR[GP1:90,2] + 29.433;
   1:L PR[91] R[100]mm/sec CNT100;
   1:  PR[GP1:91,1] = PR[GP1:90,1] + 1.580;
   1:  PR[GP1:91,2] = PR[GP1:90,2] + 28.545;
   1:L PR[91] R[100]mm/sec CNT100 TB   .50sec,CALL END_PUD;
   1:  DO[117:Laser Start]=OFF;
   1:  !Sicherheitspunkt!;
   1:  PR[92] = PR[91];
   1:  PR[92] = PR[GP1:92,3] + 50;
   1:J PR[92];
   1:  WAIT   5.00(sec);
   1:  DO[119:Gas]=OFF;
   1:  CALL HOME_ALL;
/POS
/END
